# B&R Automation Studio project CombinedLinenSoiledA9KAN (part 6)

```automation-basic
	;bDataValidFlag-> mandatory - TRUE only for last telegram as defined in CAN2 standard..
	bDataValid = FALSE 		; return data's validity status..
	endif
;******CANID421..439******T4******CANID421..439******T4******CANID421..439******T4******CANID421..439******

	;§ ID 421..439 - T4 identified -mandatories..
	if ( BIT_TST(CAN1Data.T_By1,3) AND BIT_TST(CAN1Data.T_By1,4)AND BIT_TST(CAN1Data.T_By1,5)) then

 	; a_usCustomize
		memcpy(adr(a_usOutByteArray[37]) , adr(CAN1Data.T_By0), 1)
			; im By1 liegt das Steuerbyte..
		memcpy(adr(a_usOutByteArray[38]) , adr(CAN1Data.T_By2_By3), 2)
		memcpy(adr(a_usOutByteArray[40]) , adr(CAN1Data.T_By4_By5), 2)
		memcpy(adr(a_usOutByteArray[42]) , adr(CAN1Data.T_By6_By7), 2)

	;bDataValidFlag-> mandatory - TRUE only for last telegram as defined in CAN2 standard..
	bDataValid = TRUE 		; return data's validity status..
	endif
endaction	; 421..439

;******CANID441..459************CANID441..459************CANID441..459************CANID441..459******
action 441..459:

;******CANID441..459******T1******CANID441..459******T1******CANID441..459******T1******CANID441..459******
	;§ CANID441 - T1 identified -mandatories..
; fetch By2 to get controlByte - the LOWERByte..
if(TARGETInfo_0.DataFormat = 2)then ; motorola..
	uiTemp = CAN1Data.T_By2_By3
	usTemp =  USINT(shr(uiTemp,8))
else ; i386
	usTemp = USINT(CAN1Data.T_By2_By3)
endif
	; WETCANII stamp identified.. + TelNo.1
	if ( NOT(BIT_TST(usTemp,6))AND BIT_TST(usTemp,7) ) then
;	bVorsignalFlusen
		if(BIT_TST(usTemp,0) = 1) then
			a_usOutByteArray[7] = 1
		else
			a_usOutByteArray[7] = 0
		endif
;	bSaugbeladungAktiv					1
		if(BIT_TST(usTemp,1) = 1) then
			a_usOutByteArray[8] = 1
		else
			a_usOutByteArray[8] = 0
		endif
;	bAnforderungFlusen					1
		if(BIT_TST(usTemp,2) = 1) then
			a_usOutByteArray[9] = 1
		else
			a_usOutByteArray[9] = 0
		endif
	;	uiTrocknerrestzeit
		if TARGETInfo_0.DataFormat = 2 then ; motorola
			a_usOutByteArray[0] = CAN1Data.T_By0
			a_usOutByteArray[1] = CAN1Data.T_By1
		else if TARGETInfo_0.DataFormat = 1 then ; intel
			a_usOutByteArray[0] = CAN1Data.T_By1
			a_usOutByteArray[1] = CAN1Data.T_By0
		else
		 	uiStatus = TARGETInfo_0.status
		endif
	bDataValid = FALSE ; return data's validity status..
	endif
;******CANID441..459******T2******CANID441..459******T2******CANID441..459******T2******CANID441..459******
	;§ CANID441 - T2 identified -mandatories..

	; WETCANII stamp identified.. + TelNo.2
	if (BIT_TST(usTemp,6)AND BIT_TST(usTemp,7) ) then

		memcpy(adr(a_usOutByteArray[10]), adr(CAN1Data.T_By0),2)
		memcpy(adr(a_usOutByteArray[13]), adr(CAN1Data.T_By4_By5),4)

		usTemp2 =  0
		if TARGETInfo_0.DataFormat = 2 then ; motorola
			usTemp2 = USINT(CAN1Data.T_By2_By3) ; ###HO/UM 130509 V3.3.1
 			memcpy(adr(a_usOutByteArray[12]), adr(usTemp2),1)
		else if TARGETInfo_0.DataFormat = 1 then ; intel
			usTemp2 = USINT(shr(CAN1Data.T_By2_By3,8))
			memcpy(adr(a_usOutByteArray[12]), adr(usTemp2),1)
		else
		 	uiStatus = TARGETInfo_0.status
		endif
	;bDataValidFlag-> mandatory - TRUE only for last telegram as defined in CAN2 standard..
	bDataValid = TRUE 			; return data's validity status..
	endif
endaction ; 441..459

; ###HO-250107 case mittig aufgeteilt -
elseaction:
   	uiStatus = 110
endaction
endcase
RAUS_HIER2:
if uiStatus = 110 then
	; hier weitermachen: zweiten Teil des case durchgehen
else
	; es wurde bereits ein case gefunden - raus hier..
	goto RAUS_HIER3
endif
case udCanID of

action 480:
;******CANID480******T1******CANID480******T1******CANID480******T1******CANID480******T1******CANID480******T1******
; ID 480 - T1 identified -mandatories..
	if (NOT(BIT_TST(CAN1Data.T_By0,5)) AND NOT(BIT_TST(CAN1Data.T_By0,6)) AND BIT_TST(CAN1Data.T_By0,7)) then
;------------------By 0-----------------------------
; 	bBereit
		if(BIT_TST(CAN1Data.T_By0,0) = 1) then
			a_usOutByteArray[0] = 1
		else
			a_usOutByteArray[0] = 0
		endif
; 	bBeladebereit
		if(BIT_TST(CAN1Data.T_By0,1) = 1) then
			a_usOutByteArray[2] = 1
		else
			a_usOutByteArray[2] = 0
		endif
; 	bBeladungAktiv
		if(BIT_TST(CAN1Data.T_By0,2) = 1) then
			a_usOutByteArray[3] = 1
		else
			a_usOutByteArray[3] = 0
		endif
; 	bStoerung
		if(BIT_TST(CAN1Data.T_By0,3) = 1) then
			a_usOutByteArray[4] = 1
		else
			a_usOutByteArray[4] = 0
		endif
; 	bBeladeanfHalbauto
		if(BIT_TST(CAN1Data.T_By0,4) = 1) then
			a_usOutByteArray[5] = 1
		else
			a_usOutByteArray[5] = 0
		endif
;------------------By 1-----------------------------
;	bBeladeabbruch
		if(BIT_TST(CAN1Data.T_By1,0) = 1) then
			a_usOutByteArray[7] = 1
		else
			a_usOutByteArray[7] = 0
		endif
; 	bFreigabeBeladung
		if(BIT_TST(CAN1Data.T_By1,1) = 1) then
			a_usOutByteArray[8] = 1
		else
			a_usOutByteArray[8] = 0
		endif
; 	bDurchschleusenStart
		if(BIT_TST(CAN1Data.T_By1,2) = 1) then
			a_usOutByteArray[9] = 1
		else
			a_usOutByteArray[9] = 0
		endif
;	bNotAusAero
		if(BIT_TST(CAN1Data.T_By1,3) = 1) then
			a_usOutByteArray[1] = 1
		else
			a_usOutByteArray[1] = 0
		endif
;	bBeladepause
		if(BIT_TST(CAN1Data.T_By1,4) = 1) then
			a_usOutByteArray[6] = 1
		else
			a_usOutByteArray[6] = 0
		endif
; Redundanzen b1-4
		if(BIT_TST(CAN1Data.T_By1,5) = 1) then
			a_usOutByteArray[25] = 1
		else
			a_usOutByteArray[25] = 0
		endif
		if(BIT_TST(CAN1Data.T_By1,6) = 1) then
			a_usOutByteArray[26] = 1
		else
			a_usOutByteArray[26] = 0
		endif
		if(BIT_TST(CAN1Data.T_By1,7) = 1) then
			a_usOutByteArray[27] = 1
		else
			a_usOutByteArray[27] = 0
		endif
; udPostennummer
			uiShr8 = shr(CAN1Data.T_By2_By3,8)
		a_usOutByteArray[14] = USINT(uiShr8)
		a_usOutByteArray[15] = USINT(CAN1Data.T_By2_By3)
			uiShr8 = shr(CAN1Data.T_By4_By5,8)
		a_usOutByteArray[16] = USINT(uiShr8)
		a_usOutByteArray[17] = USINT(CAN1Data.T_By4_By5)
; uiGewicht
			uiShr8 = shr(CAN1Data.T_By6_By7,8)
		a_usOutByteArray[22] = USINT(uiShr8)
		a_usOutByteArray[23] = USINT(CAN1Data.T_By6_By7)

	;bDataValidFlag-> mandatory - TRUE only for last telegram as defined in CAN2 standard..
	bDataValid = FALSE 								; return data's validity status..
	endif
;******CANID480******T2******CANID480******T2******CANID480******T2******CANID480******T2******CANID480******

	; CANID480 - T2 identified -mandatories..
	if (BIT_TST(CAN1Data.T_By0,5) AND NOT(BIT_TST(CAN1Data.T_By0,6)) AND BIT_TST(CAN1Data.T_By0,7)) then
; bProgKat
		if(BIT_TST(CAN1Data.T_By0,0) = 1) then
			a_usOutByteArray[10] = 1
		else
			a_usOutByteArray[10] = 0
		endif

; Redundanzen -> T2-By0 - bit1..4
		if(BIT_TST(CAN1Data.T_By0,1) = 1) then
			a_usOutByteArray[28] = 1
		else
			a_usOutByteArray[28] = 0
		endif
		if(BIT_TST(CAN1Data.T_By0,2) = 1) then
			a_usOutByteArray[29] = 1
		else
			a_usOutByteArray[29] = 0
		endif
		if(BIT_TST(CAN1Data.T_By0,3) = 1) then
			a_usOutByteArray[30] = 1
		else
			a_usOutByteArray[30] = 0
		endif
		if(BIT_TST(CAN1Data.T_By0,4) = 1) then
			a_usOutByteArray[31] = 1
		else
			a_usOutByteArray[31] = 0
		endif
; usReserve1
		a_usOutByteArray[24] = CAN1Data.T_By1

; uiProgKat
			uiShr8 = shr(CAN1Data.T_By2_By3,8)
		a_usOutByteArray[12] = USINT(uiShr8)
		a_usOutByteArray[13] = USINT(CAN1Data.T_By2_By3)
; udKundennummer
			uiShr8 = shr(CAN1Data.T_By4_By5,8)
		a_usOutByteArray[18] = USINT(uiShr8)
		a_usOutByteArray[19] = USINT(CAN1Data.T_By4_By5)
			uiShr8 = shr(CAN1Data.T_By6_By7,8)
		a_usOutByteArray[20] = USINT(uiShr8)
		a_usOutByteArray[21] = USINT(CAN1Data.T_By6_By7)

	;bDataValidFlag-> mandatory - TRUE only for last telegram as defined in CAN2 standard..
	bDataValid = FALSE 		; return data's validity status..
	endif
;******CANID480******T3******CANID480******T3******CANID480******T3******CANID480******T3******CANID480******

	; CANID480 - T3 identified -mandatories..
	if (NOT(BIT_TST(CAN1Data.T_By0,5)) AND BIT_TST(CAN1Data.T_By0,6) AND BIT_TST(CAN1Data.T_By0,7)) then

	; Redundanzen -> T3-By0 - bit1..2 - bit3..4 nicht verwendet..
		if(BIT_TST(CAN1Data.T_By0,0) = 1) then
			a_usOutByteArray[32] = 1
		else
			a_usOutByteArray[32] = 0
		endif
		if(BIT_TST(CAN1Data.T_By0,1) = 1) then
			a_usOutByteArray[33] = 1
		else
			a_usOutByteArray[33] = 0
		endif

	; a_usCustomize
		memcpy(adr(a_usOutByteArray[34]) , adr(CAN1Data.T_By1), 1)
		memcpy(adr(a_usOutByteArray[35]) , adr(CAN1Data.T_By2_By3), 2)
		memcpy(adr(a_usOutByteArray[37]) , adr(CAN1Data.T_By4_By5), 2)
		memcpy(adr(a_usOutByteArray[39]) , adr(CAN1Data.T_By6_By7), 2)

	;bDataValidFlag-> mandatory - TRUE only for last telegram as defined in CAN2 standard..
	bDataValid = TRUE 		; return data's validity status..
	endif
endaction ; 480

action 481:
;******CANID481******T1******CANID481******T1******CANID481******T1******CANID481******T1******CANID481******T1******
; ID 481 - T1 identified -mandatories..
	if (NOT(BIT_TST(CAN1Data.T_By0,5)) AND NOT(BIT_TST(CAN1Data.T_By0,6)) AND BIT_TST(CAN1Data.T_By0,7)) then

; bBereit
		if(BIT_TST(CAN1Data.T_By0,0) = 1) then
			a_usOutByteArray[0] = 1
		else
			a_usOutByteArray[0] = 0
		endif
; bBeladeanfAuto
		if(BIT_TST(CAN1Data.T_By0,1) = 1) then
			a_usOutByteArray[2] = 1
		else
			a_usOutByteArray[2] = 0
		endif
; bStoerung
		if(BIT_TST(CAN1Data.T_By0,2) = 1) then
			a_usOutByteArray[3] = 1
		else
			a_usOutByteArray[3] = 0
		endif
; bAnlagenstrgHalbauto
		if(BIT_TST(CAN1Data.T_By0,3) = 1) then
			a_usOutByteArray[4] = 1
		else
			a_usOutByteArray[4] = 0
		endif
; bAnlagenStrgAuto
		if(BIT_TST(CAN1Data.T_By0,4) = 1) then
			a_usOutByteArray[5] = 1
		else
			a_usOutByteArray[5] = 0
		endif
; Redundanzen b1-4
		if(BIT_TST(CAN1Data.T_By1,4) = 1) then
			a_usOutByteArray[23] = 1
		else
			a_usOutByteArray[23] = 0
		endif
		if(BIT_TST(CAN1Data.T_By1,5) = 1) then
			a_usOutByteArray[24] = 1
		else
			a_usOutByteArray[24] = 0
		endif
		if(BIT_TST(CAN1Data.T_By1,6) = 1) then
			a_usOutByteArray[25] = 1
		else
			a_usOutByteArray[25] = 0
		endif
		if(BIT_TST(CAN1Data.T_By1,7) = 1) then
			a_usOutByteArray[26] = 1
		else
			a_usOutByteArray[26] = 0
		endif
; bDurchschleusen
		if(BIT_TST(CAN1Data.T_By1,0) = 1) then
			a_usOutByteArray[7] = 1
		else
			a_usOutByteArray[7] = 0
		endif
; bFreigabeDurchschl
		if(BIT_TST(CAN1Data.T_By1,1) = 1) then
			a_usOutByteArray[8] = 1
		else
			a_usOutByteArray[8] = 0
		endif
; bNotAusAnlagenStrg
		if(BIT_TST(CAN1Data.T_By1,2) = 1) then
			a_usOutByteArray[1] = 1
		else
			a_usOutByteArray[1] = 0
		endif
; bPauseAktiv
		if(BIT_TST(CAN1Data.T_By1,3) = 1) then
			a_usOutByteArray[6] = 1
		else
			a_usOutByteArray[6] = 0
		endif
; udPostennummer
			uiShr8 = shr(CAN1Data.T_By2_By3,8)
		a_usOutByteArray[18] = USINT(uiShr8)
		a_usOutByteArray[19] = USINT(CAN1Data.T_By2_By3)
			uiShr8 = shr(CAN1Data.T_By4_By5,8)
		a_usOutByteArray[20] = USINT(uiShr8)
		a_usOutByteArray[21] = USINT(CAN1Data.T_By4_By5)
; uiGewicht
			uiShr8 = shr(CAN1Data.T_By6_By7,8)
		a_usOutByteArray[12] = USINT(uiShr8)
		a_usOutByteArray[13] = USINT(CAN1Data.T_By6_By7)

	;bDataValidFlag-> mandatory - TRUE only for last telegram as defined in CAN2 standard..
	bDataValid = FALSE 								; return data's validity status..

	endif
;******CANID481******T2******CANID481******T2******CANID481******T2******CANID481******T2******CANID481******

	; CANID481 - T2 identified -mandatories..
	if (BIT_TST(CAN1Data.T_By0,5) AND NOT(BIT_TST(CAN1Data.T_By0,6)) AND BIT_TST(CAN1Data.T_By0,7)) then
; bProgKat
		if(BIT_TST(CAN1Data.T_By0,0) = 1) then
			a_usOutByteArray[9] = 1
		else
			a_usOutByteArray[9] = 0
		endif
; Redundanzen T2By0 /b6-10
		if(BIT_TST(CAN1Data.T_By0,1) = 1) then
			a_usOutByteArray[27] = 1
		else
			a_usOutByteArray[27] = 0
		endif
		if(BIT_TST(CAN1Data.T_By0,2) = 1) then
			a_usOutByteArray[28] = 1
		else
			a_usOutByteArray[28] = 0
		endif
		if(BIT_TST(CAN1Data.T_By0,3) = 1) then
			a_usOutByteArray[29] = 1
		else
			a_usOutByteArray[29] = 0
		endif
		if(BIT_TST(CAN1Data.T_By0,4) = 1) then
			a_usOutByteArray[30] = 1
		else
			a_usOutByteArray[30] = 0
		endif
; usReserve1
		a_usOutByteArray[22] = CAN1Data.T_By1
; uiProgKat
			uiShr8 = shr(CAN1Data.T_By2_By3,8)
		a_usOutByteArray[10] = USINT(uiShr8)
		a_usOutByteArray[11] = USINT(CAN1Data.T_By2_By3)
; udKundennummer
			uiShr8 = shr(CAN1Data.T_By4_By5,8)
		a_usOutByteArray[14] = USINT(uiShr8)
		a_usOutByteArray[15] = USINT(CAN1Data.T_By4_By5)
			uiShr8 = shr(CAN1Data.T_By6_By7,8)
		a_usOutByteArray[16] = USINT(uiShr8)
		a_usOutByteArray[17] = USINT(CAN1Data.T_By6_By7)

	;bDataValidFlag-> mandatory - TRUE only for last telegram as defined in CAN2 standard..
	bDataValid = FALSE 		; return data's validity status..
	endif

;******CANID481******T3******CANID481******T3******CANID481******T3******CANID481******T3******CANID481******

	; CANID481 - T3 identified -mandatories..
	if (NOT(BIT_TST(CAN1Data.T_By0,5)) AND BIT_TST(CAN1Data.T_By0,6) AND BIT_TST(CAN1Data.T_By0,7)) then

	; Redundanzen bR9..10
		if(BIT_TST(CAN1Data.T_By0,1) = 1) then
			a_usOutByteArray[31] = 1
		else
			a_usOutByteArray[31] = 0
		endif
		if(BIT_TST(CAN1Data.T_By0,2) = 1) then
			a_usOutByteArray[32] = 1
		else
			a_usOutByteArray[32] = 0
		endif

	; a_usCustomize
		memcpy(adr(a_usOutByteArray[33]) , adr(CAN1Data.T_By1), 1)
		memcpy(adr(a_usOutByteArray[34]) , adr(CAN1Data.T_By2_By3), 2)
		memcpy(adr(a_usOutByteArray[36]) , adr(CAN1Data.T_By4_By5), 2)
		memcpy(adr(a_usOutByteArray[38]) , adr(CAN1Data.T_By6_By7), 2)

	;bDataValidFlag-> mandatory - TRUE only for last telegram as defined in CAN2 standard..
	bDataValid = TRUE 		; return data's validity status..
	endif
endaction ; 481

;********************************************************************************************************
;********************************************************************************************************
; add new Obj types here..
;********************************************************************************************************
;********************************************************************************************************

elseaction:
	uiStatus = 110
endaction

endcase ; udCanID

RAUS_HIER3:

END_FUNCTION_BLOCK
```

#### _Seti386CAN2TypeToCAN1Type.ab
```automation-basic
FUNCTION_BLOCK _Seti386CAN2TypeToCAN1Type
;********************************************************************************************************
; * Implementation of _Seti386CAN2TypeToCAN1Type
;********************************************************************************************************
; * version 		1.1.0
; * last change		sep, 12th, 2005
; * by				H.O.
;********************************************************************************************************
;********************************************************************************************************
; 	-> 	pCAN2Data			.. pointer to CAN2 structure that contains data to read or write
; 	-> 	iTelegramIndex		.. telegram index exctractet from received / broadcasted telegram
; 		pCAN1Data 		->	.. return the address of CAN1 struct
;********************************************************************************************************
; V1.1.0 ###HO  - 120905
;	* 5th tel added
;********************************************************************************************************

; set local pointer to incoming CAN2 uni structure
pLocalCAN2UniData access (pCAN2Data)
LocalCAN2UniData = pLocalCAN2UniData

; create CAN1 telegram from CAN2 te structure passed in..
case iTelegramIndex of

	action 1:
		LocalCAN1Data.T_By0 	= LocalCAN2UniData.T1_By0
		LocalCAN1Data.T_By1 	= LocalCAN2UniData.T1_By1

		uiShiftUPPERWord 		= shr(LocalCAN2UniData.T1_By2_By3,8) ; move UPPER byte to the right
		uiShiftLOWERWord 		= shl(LocalCAN2UniData.T1_By2_By3,8) ; move LOWER byte to the left
		LocalCAN1Data.T_By2_By3 = uiShiftUPPERWord + uiShiftLOWERWord ; now uiShiftWord contains LocalCAN2UniData.T1_By2_By3 in reverse order

		uiShiftUPPERWord 		= shr(LocalCAN2UniData.T1_By4_By5,8) ; move UPPER byte to the right
		uiShiftLOWERWord 		= shl(LocalCAN2UniData.T1_By4_By5,8) ; move LOWER byte to the left
		LocalCAN1Data.T_By4_By5 = uiShiftUPPERWord + uiShiftLOWERWord ; now uiShiftWord contains LocalCAN2UniData.T1_By2_By3 in reverse order

		uiShiftUPPERWord 		= shr(LocalCAN2UniData.T1_By6_By7,8) ; move UPPER byte to the right
		uiShiftLOWERWord 		= shl(LocalCAN2UniData.T1_By6_By7,8) ; move LOWER byte to the left
		LocalCAN1Data.T_By6_By7 = uiShiftUPPERWord + uiShiftLOWERWord ; now uiShiftWord contains LocalCAN2UniData.T1_By2_By3 in reverse order
	endaction
		action 2:
		LocalCAN1Data.T_By0 	= LocalCAN2UniData.T2_By0
		LocalCAN1Data.T_By1 	= LocalCAN2UniData.T2_By1

		uiShiftUPPERWord 		= shr(LocalCAN2UniData.T2_By2_By3,8) ; move UPPER byte to the right
		uiShiftLOWERWord 		= shl(LocalCAN2UniData.T2_By2_By3,8) ; move LOWER byte to the left
		LocalCAN1Data.T_By2_By3 = uiShiftUPPERWord + uiShiftLOWERWord ; now uiShiftWord contains LocalCAN2UniData.T1_By2_By3 in reverse order

		uiShiftUPPERWord 		= shr(LocalCAN2UniData.T2_By4_By5,8) ; move UPPER byte to the right
		uiShiftLOWERWord 		= shl(LocalCAN2UniData.T2_By4_By5,8) ; move LOWER byte to the left
		LocalCAN1Data.T_By4_By5 = uiShiftUPPERWord + uiShiftLOWERWord ; now uiShiftWord contains LocalCAN2UniData.T1_By2_By3 in reverse order

		uiShiftUPPERWord 		= shr(LocalCAN2UniData.T2_By6_By7,8) ; move UPPER byte to the right
		uiShiftLOWERWord 		= shl(LocalCAN2UniData.T2_By6_By7,8) ; move LOWER byte to the left
		LocalCAN1Data.T_By6_By7 = uiShiftUPPERWord + uiShiftLOWERWord ; now uiShiftWord contains LocalCAN2UniData.T1_By2_By3 in reverse order
	endaction
		action 3:
		LocalCAN1Data.T_By0 	= LocalCAN2UniData.T3_By0
		LocalCAN1Data.T_By1 	= LocalCAN2UniData.T3_By1

		uiShiftUPPERWord 		= shr(LocalCAN2UniData.T3_By2_By3,8) ; move UPPER byte to the right
		uiShiftLOWERWord 		= shl(LocalCAN2UniData.T3_By2_By3,8) ; move LOWER byte to the left
		LocalCAN1Data.T_By2_By3 = uiShiftUPPERWord + uiShiftLOWERWord ; now uiShiftWord contains LocalCAN2UniData.T1_By2_By3 in reverse order

		uiShiftUPPERWord 		= shr(LocalCAN2UniData.T3_By4_By5,8) ; move UPPER byte to the right
		uiShiftLOWERWord 		= shl(LocalCAN2UniData.T3_By4_By5,8) ; move LOWER byte to the left
		LocalCAN1Data.T_By4_By5 = uiShiftUPPERWord + uiShiftLOWERWord ; now uiShiftWord contains LocalCAN2UniData.T1_By2_By3 in reverse order

		uiShiftUPPERWord 		= shr(LocalCAN2UniData.T3_By6_By7,8) ; move UPPER byte to the right
		uiShiftLOWERWord 		= shl(LocalCAN2UniData.T3_By6_By7,8) ; move LOWER byte to the left
		LocalCAN1Data.T_By6_By7 = uiShiftUPPERWord + uiShiftLOWERWord ; now uiShiftWord contains LocalCAN2UniData.T1_By2_By3 in reverse order
	endaction
		action 4:
		LocalCAN1Data.T_By0 	= LocalCAN2UniData.T4_By0
		LocalCAN1Data.T_By1 	= LocalCAN2UniData.T4_By1

		uiShiftUPPERWord 		= shr(LocalCAN2UniData.T4_By2_By3,8) ; move UPPER byte to the right
		uiShiftLOWERWord 		= shl(LocalCAN2UniData.T4_By2_By3,8) ; move LOWER byte to the left
		LocalCAN1Data.T_By2_By3 = uiShiftUPPERWord + uiShiftLOWERWord ; now uiShiftWord contains LocalCAN2UniData.T1_By2_By3 in reverse order

		uiShiftUPPERWord 		= shr(LocalCAN2UniData.T4_By4_By5,8) ; move UPPER byte to the right
		uiShiftLOWERWord 		= shl(LocalCAN2UniData.T4_By4_By5,8) ; move LOWER byte to the left
		LocalCAN1Data.T_By4_By5 = uiShiftUPPERWord + uiShiftLOWERWord ; now uiShiftWord contains LocalCAN2UniData.T1_By2_By3 in reverse order

		uiShiftUPPERWord 		= shr(LocalCAN2UniData.T4_By6_By7,8) ; move UPPER byte to the right
		uiShiftLOWERWord 		= shl(LocalCAN2UniData.T4_By6_By7,8) ; move LOWER byte to the left
		LocalCAN1Data.T_By6_By7 = uiShiftUPPERWord + uiShiftLOWERWord ; now uiShiftWord contains LocalCAN2UniData.T1_By2_By3 in reverse order
	endaction
	action 5:
		LocalCAN1Data.T_By0 	= LocalCAN2UniData.T5_By0
		LocalCAN1Data.T_By1 	= LocalCAN2UniData.T5_By1

		uiShiftUPPERWord 		= shr(LocalCAN2UniData.T5_By2_By3,8) ; move UPPER byte to the right
		uiShiftLOWERWord 		= shl(LocalCAN2UniData.T5_By2_By3,8) ; move LOWER byte to the left
		LocalCAN1Data.T_By2_By3 = uiShiftUPPERWord + uiShiftLOWERWord ; now uiShiftWord contains LocalCAN2UniData.T1_By2_By3 in reverse order

		uiShiftUPPERWord 		= shr(LocalCAN2UniData.T5_By4_By5,8) ; move UPPER byte to the right
		uiShiftLOWERWord 		= shl(LocalCAN2UniData.T5_By4_By5,8) ; move LOWER byte to the left
		LocalCAN1Data.T_By4_By5 = uiShiftUPPERWord + uiShiftLOWERWord ; now uiShiftWord contains LocalCAN2UniData.T1_By2_By3 in reverse order

		uiShiftUPPERWord 		= shr(LocalCAN2UniData.T5_By6_By7,8) ; move UPPER byte to the right
		uiShiftLOWERWord 		= shl(LocalCAN2UniData.T5_By6_By7,8) ; move LOWER byte to the left
		LocalCAN1Data.T_By6_By7 = uiShiftUPPERWord + uiShiftLOWERWord ; now uiShiftWord contains LocalCAN2UniData.T1_By2_By3 in reverse order
	endaction
endcase

; pass pointer to CAN1 telegram to output..
pCAN1Data = ADR(LocalCAN1Data)

;********************************************************************************************************
;********************************************************************************************************
END_FUNCTION_BLOCK
```

#### _swapUINT.ab
```automation-basic
FUNCTION _swapUINT
;*************************************************************************************
(* Implementation of _swapUINT *)
;*************************************************************************************
;  Identisch CONVERT::swapUINT -die macht aber Streit beim Wechsel zw. m68k und i386 !
;*************************************************************************************
usHIGHERBYTE = USINT(shr(uiIn,8))
usLOWERBYTE  = USINT(uiIn)

_swapUINT = usLOWERBYTE*256 + usHIGHERBYTE
;*************************************************************************************
END_FUNCTION
```

#### _version.ab
```automation-basic
FUNCTION_BLOCK _version
;******************************************************************
(* Implementation of _version *)
;******************************************************************
strcpy(adr(szVersion ),"V3.6.2")
uiBuild = 00000 ;  - 170112 - 1230
;******************************************************************
; History
; -------
; V3.6.2 - ###HO - 170112
;	*  Korrektur COB306.uiGew /.bUebergabest /.bNotAusAero
;	*  Korrektur COB316.bBereit
;	*  Korrektur COB371.a_usCustom /.bBereit
; V3.6.1 - ###HO - 160112
;	*  Korrektur: Letztes Einzeltel. 306,316,361..,371.. ohne Inhalt
;		* COB306 Uebergabestörung++ / a_usCustomize++ lt. TIS 2003-07g V1.1.0
;		* COB316 a_usCustomize++ lt. TIS 2003-07g V1.1.0
;		* 361..369 a_uscustomize++ / bBereit ++ lt. TIS 2003-07k V1.1.0
;		* 371..379 a_uscustomize++ / bBereit ++ lt. TIS 2003-07k V1.1.0
; V3.6.0 - ###HO - 120210
;	* COB120 auch für ID 150,160,170,180,190
;	* COB121 auch für ID 151,161,171,181,191
; V3.5.0 - ###HO - 050210
;	* COB301.Entladeueberwachung ++
; V3.4.0 - ###HO - 211209
;	* COB 110 + 111 neu (Test i386 ok, todo: m68k)
; V3.3.2 - ###HO - 130509
;	* WARNUNGEN nicht verw. Var entfernt
; V3.3.1 - ###HO - 130509
;	* SetCAN1TypeToByteArray::Korrektur 4x Compilerwarnung durch BuR UM
; V3.3.0 - ###HO - 140409
;	* COB311.StartPresse
;	* COB211.SicherhTuer
;	* COB211.StartbefAnPT
; V3.2.3 - ###HO - 070308
; 	* COB301.LS_Bandende ++
; 	* COB301.bNotAus --
; 	* COB311.SchutzgitterOffen ++
; 	* COB252.SperreBereich ++
; V3.2.2 - ###HO - 111007
; 	* _SetCAN2COBTypeToCAN2Type::COB211.usFehlerZweiteEW
; 	* _SetCAN1TypeToByteArray:: Korrektur Lesen von 211.bStartDesinfektion, 211.bStartSpuelen, 211.bEndeSpuelen
; V3.2.1 - ###hcs/HO - 101007
; 	COB_ID130und140 und COB_ID131und141 entfernt - stattdessen Neudefinition:
; 		* COB 130 und COB140 wie COB120
;		* COB131 und COB141 wie COB121
; V3.2.0 - ###HO - 040907
;	* COB251.bBeladestart
;		* _SetCAN2COBTypeToCAN2Type
;		* _SetCAN1TypeToByteArray
;		* _ConvertDataToi386
;	* COBs 261,262 hinzugefügt
; 	* neu: COB301bis304, COB311bis314, COB251u253u255, COB252u254u256, COB351bis354
;	* obsolet/umbenannt (s.o.): COB301, COB351, COB251, COB252
; V3.1.2 - ###HO - 250107
;	* _SetCAN2COBTypeToCAN2Type + _SetCAN1TypeToByteArray ::Sprung >32k (MyCheck) beseitigt
; V3.1.1 - ###HO - 110107
;	* _SetCAN2COBTypeToCAN2Type:351 lt. TIS 07j)-V1.4.3
; V3.1.0 - ###HO - 141206
;	* COBs 126,128 (=COB120) und 127,129 (=COB121) hinzugefügt
; V3.0.9 - ###HO - 260106
;	* _SetCAN2COBTypeToCAN2Type + _SetCAN1TypeToByteArray::COB231.Reserve1+2
; V3.0.8 - ###HO - 21.11.2005
;	* _SetCAN2COBTypeToCAN2Type::LocalCOB_Typ_251 -> LocalCOB_Typ_253,LocalCOB_Typ_255,LocalCOB_Typ_257
; V3.0.7 - ###HO - 17.11.2005
;	* Read:COB251=253=255=257
;	* Wrt: COB252=254=256=258
;	* _GetNumberOfCan1Tels::COB254,256,258:: 2->3
;	* _SetCAN2COBTypeToCAN2Type::COB253,255,257::LocalCAN2Data.T2_By0,4
; V3.0.6 - ###HO - 21.10.2005
;	* _SetCAN2COBTypeToCAN2Type::COB_ID421bis439 erweitert für IDs 422..439
; V3.0.5 - ###HO - 14.10.2005
;	* _SetCAN1TypeToByteArray::COB201.uiProgrammKategorie - Alignmentbyte auf xx[5]..
; V3.0.4 - ###HO - 06.10.2005
; 	* a_usCustomize für COBs 301,311,221,231,201,211,209,219
; V3.0.3 - ###HO - 05.10.2005
;	* COB_ID211.bSchiebeimpulsWETShuttle ersetzt durch bSchiebeimpSpbPreXOR_WETShuttle lt. TIS 2003_07c) V1.1.1
; V3.0.2 - ###HO - 19.09.2005
;	* Can2Init().doMemType
; V3.0.0 - ###HO - 12.09.2005
;	* COBxxx.a_usCustomize[0..6] hinzugefügt
;	* COBs 307+317 neu
; V2.1.5 - ###HO - 31.08.2005
;	* Ergänzung Hilfe COB441
;	* Aktualisierung Datentypen ‚COB_ID401bis419’ + ‚COB_ID441bis459’ TIS2003-7h nach V1.2.2b
;V2.1.4 ###HO - 17.02.2005
;·      CAN2Init(): ‚20613’ für ‚usUniqueIDCAN2Init’ > 9
; V2.1.3 ###HO - 110205
; 	* '_SetCAN1TypeToByteArray':: Autoerkennung: Lesen COB120::2oder4Tels
; 	* 'CAN2RW':: Autoerkennung: Schreiben COB120::2oder4Tels
; V2.1.2 ###HO - 070205
;	* V2.1.1 auch für m68k
; V2.1.1 ###HO
; 	* Korrektur Bezeichner szCAN2Write/ReadDO für DatObjCreate() - sonst status '20601'
;	* Speicher für DOs nach Warmstart wurde nicht wieder freigegeben
;		-> Instanzenabhängige Generierung von DOs anhand UniqueCAN2Init-Handle
; V2.1.0 ###HO	150404
;	* Redundancy support done for COBs: 480,481
; 	* COB130.udKundenummer korrigiert
;	* COB201 Desinfektion ergänzt
;		* bFreigabeDesinfektion, bTankIstLeer, bFreigabeSpuelen, EndeDesinfektion
;	* COB211 Desinfektion ergänzt + bSchiebeimpuls in bSchiebeimpulsWETShuttle umbenannt
;		* bSchiebeimpulsZweiteEntwaess korrigiert
;		* bStartDesinfektion,bEndeSpuelen,bStartSpuelen	hinzugefügt
;	* COB401..419
;		* bProgrammabbruch umbenannt in bVorsignal
;		* bKippsperre ergänzt
;	* COB 421..439
;		* 'bEntlaedt' umbenannt in 'bEntlade'
;		* 'bNotAus' umbenannt in 'bNotAusTrockner
; 	* COB231
;		* usEntladungTrockner 	-> By2 + usTransferZBvorHFB			-> By3
;		* usFehlernummer 		-> By4 +  usTransferZBvorTrockner 	-> By5
;	* COB441..459 hinzugefügt
;	* DO "AdrIC2Prot" replaced by pCAN2Init_ident
;	* enable added
;	* Instance individual DOs generated (!)- mandatory for support of same CANIDs on different CANIFs..
; V 2.0.0 ###HO
;		* COBs 123, 251,252,480,481 added
; 		* COB 122 replaced
; 		* COBs 120,121 modified
; 		* COB 122 number of tels changed from two to four
;		* manually passed size of CANQueue removed - Queuesize always is four now..
; 		* DO "AdrIC2Prot" added to replace OutPara 'p_InitCAN2Protocol'
;		* InPara 'p_InitCAN2Protocol' replaced by DO 'AdrIC2Prot'
; 		* Communication-globalPara 'CAN2Init.iMode' replaced by COB-individual-parameter 'InitCAN2PV.iMode'
; 		* mode by that telegrams have been sent within cycletime changed:
;		* 200ms - exclusively between tels with identical CANID
; 		* all tels of WETCAN2Tel are sent immediately
; V1.00 ###HO -	071003
;		* erste Version
;******************************************************************

END_FUNCTION_BLOCK
```

#### CAN2Init.ab
```automation-basic
FUNCTION_BLOCK CAN2Init
;********************************************************************************************************
;* Implementation of CAN2Init
;********************************************************************************************************
; * version 		3.0.2
; * last change		sep, 19th, 2005
; * by				H.O.
;********************************************************************************************************
; * History:
;***********
; * 3.0.2 	###HO - 190905
; 	* IN doMemType anstatt doUSRRAM
; * V2.1.2	###HO - 070205
;	* V2.1.1 auch für m68k
; * V2.1.1
; 	* Korrektur Bezeichner szCAN2Write/ReadDO für DatObjCreate() - sonst status '20601'
;	* Speicher für DOs nach Warmstart wurde nicht wieder freigegeben
;		-> Instanzenabhängige Generierung von DOs anhand UniqueCAN2Init-Handle
; * V2.1.0
;		* DO "AdrIC2Prot" replaced by pCAN2Init_ident
;		* enable added
;		* instance individual DOs generated
; 			-> mandatory for support of same CANIDs on different CANIFs..
; * V 1.0.0		-> 1st version for AS..
; * V 2.0.0
;		* manually passed size of CANQueue removed - Queuesize always is four now..
; 		* DO "AdrIC2Prot" added to replace OutPara 'p_InitCAN2Protocol'
;********************************************************************************************************
;********************************************************************************************************

if (enable = 0) then
	goto ENDE
endif

; initiate return status of CAN2Init()
uiStatus = 0;  105 ;

; generate identifier for InitDO ...
strcpy(ADR(szInitDO),"CAN2Ini") ; ###HO - 170205 - verkürzt - sonst '20613'
usInitDOInstanceNumber = usUniqueIDCAN2Init
itoa(DINT(usInitDOInstanceNumber), adr(szInitDOInstanceNumber))
; ###HO300904 - "CAN2Init1"
strcat(ADR(szInitDO), adr(szInitDOInstanceNumber))

; create DO with R/W info..
DatObjCreate_InitDO.enable	= 1
DatObjCreate_InitDO.grp		= 0
DatObjCreate_InitDO.pName	= ADR(szInitDO) ; "CAN2Init1"
DatObjCreate_InitDO.len		= uiNumberOfCAN2COBs * sizeof(Local_InitCAN2PV) ; size of DO depends on number of COBs..
DatObjCreate_InitDO.MemType	= doMemType ; doUSRRAM 	; = usrram ist warmstartsicher(!)
DatObjCreate_InitDO.Option	= 1 		; 1-> no crc check..
DatObjCreate_InitDO.pCpyData = adr(pStartAdrDO)	; not in use..
DatObjCreate_InitDO FUB DatObjCreate()
if((uiStatus = 0) and (DatObjCreate_InitDO.status <> 20601))  then
	uiStatus = DatObjCreate_InitDO.status
endif

DatObjInfo(1, ADR(szInitDO), DO_StatInfo, DO_ID, DO_StartAdr, DO_Len, DO_Memtype, DO_Option, DO_ChangeDat )
;***************************************************************************************
; generate identifier for InitDO ...
strcpy(ADR(szCAN2WriteDO),"CAN2Wrt") ; ###HO - 170205 - verkürzt - sonst '20613'
itoa(DINT(usInitDOInstanceNumber), adr(szInitDOInstanceNumber))
;###HO 300904 - strcat('szInitDO',,)
strcat(ADR(szCAN2WriteDO), adr(szInitDOInstanceNumber)) ; addInstNumber to szCAN2WriteDO

DatObjCreate_WriteDO.enable		= 1
DatObjCreate_WriteDO.grp		= 0
DatObjCreate_WriteDO.pName		= adr(szCAN2WriteDO) ; "CAN2Write"
DatObjCreate_WriteDO.len		= uiNumberOfCAN2COBs * sizeof(CAN2Write)
DatObjCreate_WriteDO.MemType	= doMemType ; doUSRRAM
DatObjCreate_WriteDO.Option		= 1
DatObjCreate_WriteDO.pCpyData	= adr(pStartAdrDOCAN2Write)
DatObjCreate_WriteDO FUB DatObjCreate()
if((uiStatus = 0) and (DatObjCreate_WriteDO.status <> 20601))  then
	uiStatus = DatObjCreate_WriteDO.status
endif
DatObjInfo(1, ADR(szCAN2WriteDO), DO_StatInfo, DO_IDCAN2Write, DO_StartAdr, DO_Len, DO_Memtype, DO_Option, DO_ChangeDat )
;***************************************************************************************

; generate identifier for InitDO ...
strcpy(ADR(szCAN2ReadDO),"CAN2Rd") ; ###HO - 170205 - verkürzt - sonst '20613'
itoa(DINT(usInitDOInstanceNumber), adr(szInitDOInstanceNumber))
;###HO 300904 - strcat('szInitDO',,)
strcat(ADR(szCAN2ReadDO), adr(szInitDOInstanceNumber)) ; addInstNumber to szCAN2ReadDO

DatObjCreate_ReadDO.enable		= 1
DatObjCreate_ReadDO.grp			= 0
DatObjCreate_ReadDO.pName		= ADR(szCAN2ReadDO)
DatObjCreate_ReadDO.len			= uiNumberOfCAN2COBs * sizeof(CAN2Read)
DatObjCreate_ReadDO.MemType		= doMemType ; doUSRRAM
DatObjCreate_ReadDO.Option		= 1
DatObjCreate_ReadDO.pCpyData	= adr(pStartAdrDOCAN2Read)
DatObjCreate_ReadDO FUB DatObjCreate()
if((uiStatus = 0) and (DatObjCreate_ReadDO.status <> 20601))  then
	uiStatus = DatObjCreate_ReadDO.status
endif
DatObjInfo(1, adr(szCAN2ReadDO), DO_StatInfo, DO_IDCAN2Read, DO_StartAdr, DO_Len, DO_Memtype, DO_Option, DO_ChangeDat )

;********************************************
; prepare writing to DO
DatObjWrite_InitDO.enable	= 1							; wanna write to DO..
DatObjWrite_InitDO.ident	= DO_ID						; from DOInfo..
DatObjWrite_InitDO.len		= sizeof(Local_InitCAN2PV) 	; size of single DO - former LocalCAN2InitData
;********************************************
DatObjWrite_WriteDO.enable	= 1
DatObjWrite_WriteDO.ident	= DO_IDCAN2Write
DatObjWrite_WriteDO.len		= sizeof(CAN2Write)
;********************************************
DatObjWrite_ReadDO.enable	= 1
DatObjWrite_ReadDO.ident	= DO_IDCAN2Read
DatObjWrite_ReadDO.len		= sizeof(CAN2Read)
;********************************************

; CANOpen() sufficent for CANrd() + CANqwrite()
CANopen_0.enable	= 1
CANopen_0.baud_rate	= 25
CANopen_0.cob_anz	= uiNumberOfCAN2COBs *2
CANopen_0.error_adr	= ADR(ErrAdrNotInUse)
CANopen_0.device	= ADR(szCANInterface)
CANopen_0.info		= 0 ; don't use extd mode of CANCtrl ..
CANopen_0 FUB CANopen()
if(uiStatus = 0) then
	uiStatus = CANopen_0.status
endif
;********************************************

; now -fill DOs with necessarily data
loop iLoopIdx = 0 to (uiNumberOfCAN2COBs -1) do
	memcpy(adr(LocalInitCAN2PV), (pInitCAN2PV + sizeof(LocalInitCAN2PV)*iLoopIdx), sizeof(LocalInitCAN2PV))

	; pass 'InitData' -> '_InitData' ..
	Local_InitCAN2PV.pPVData			= LocalInitCAN2PV.pPVData
	Local_InitCAN2PV.uiObjNr			= LocalInitCAN2PV.uiCANID
	Local_InitCAN2PV.usCommDirection	= LocalInitCAN2PV.usCommDirection
	Local_InitCAN2PV.pEvVar				= LocalInitCAN2PV.pEvVar
	Local_InitCAN2PV.uiCOB_ident		= UINT(iLoopIdx + 900) 	; internal identifier - not in use
	Local_InitCAN2PV.bRunning			= FALSE 				; not in use
	; from V1.1.0 -> COB-individual selection of mode..
	Local_InitCAN2PV.iMode				= LocalInitCAN2PV.iMode

	; check CommDirection to decide whether to initiate a CANqueue() ..
	; initiate for all read operations single CANqueue  - establishing CANQueue only in read direction necessary..
	if (LocalInitCAN2PV.usCommDirection = 0) then		; read to COB..

		; initiate CANqueue for read operation..
		CANqueue_0.enable	= 1
		CANqueue_0.us_ident	= CANopen_0.us_ident
		CANqueue_0.can_id	= LocalInitCAN2PV.uiCANID
		; uiCANqueueSize from V1.0.0 removed -> set to max count of single tels..
		CANqueue_0.size		= 5 ; telegram capacity of queue..
		CANqueue_0 FUB CANqueue()
		if(uiStatus = 0) then
			uiStatus = CANqueue_0.status
			exitif (CANqueue_0.status <> 0)
		endif

		_GetNumberOfCan1Tels_0.pPV		= Local_InitCAN2PV.pPVData
		_GetNumberOfCan1Tels_0.uiObjNr	= Local_InitCAN2PV.uiObjNr
		_GetNumberOfCan1Tels_0 FUB _GetNumberOfCan1Tels()

		; uiCAN_q_ident isn't passed in by user -> created by CANqueue ..
		Local_InitCAN2PV.udCAN_q_ident	= CANqueue_0.q_ident ;

		; write uiObjNr to DO..
		CAN2Read.uiObjNr				= Local_InitCAN2PV.uiObjNr
		CAN2Read.iNumberOfTels			= _GetNumberOfCan1Tels_0.iNumberOfCan1Tels
		CAN2Read.iNumberReceivedTels	= 0

		; reset data of WriteDO
		CAN2Write.bBusy 			= FALSE
		CAN2Write.iNumberOfTels 	= 0
		CAN2Write.iTelsSent			= 0
		CAN2Write.tTimeLastTelSent 	= TIME(0)
		CAN2Write.uiCOB_ident		= iLoopIdx + 900

	else if (LocalInitCAN2PV.usCommDirection = 1) then	; COB is defined as to 'write'
		Local_InitCAN2PV.udCAN_q_ident	= 0	; object to write - no queue established

		; establish DO with CAN2Data of COBs to write..
		_GetNumberOfCan1Tels_0.pPV		= Local_InitCAN2PV.pPVData
		_GetNumberOfCan1Tels_0.uiObjNr	= Local_InitCAN2PV.uiObjNr
		_GetNumberOfCan1Tels_0 FUB _GetNumberOfCan1Tels()

		_SetCAN2COBTypeToCAN2Type_0.p_InitCAN2PV = adr(Local_InitCAN2PV)
		_SetCAN2COBTypeToCAN2Type_0 FUB _SetCAN2COBTypeToCAN2Type()
		; don't read PVs now- actualize process images at runtime..
		; memcpy(adr(CAN2Write.CAN2), _SetCAN2COBTypeToCAN2Type_0.pCAN2DtaUni, sizeof(CAN2Write.CAN2))

		CAN2Write.bBusy 			= FALSE
		CAN2Write.iNumberOfTels 	= _GetNumberOfCan1Tels_0.iNumberOfCan1Tels
		CAN2Write.iTelsSent			= 0
		CAN2Write.tTimeLastTelSent 	= TIME(0)
		CAN2Write.uiCOB_ident		= iLoopIdx + 900

			; reset content of DORead
			CAN2Read.uiObjNr = 0
			loop iLoopIdxTemp = 0 to 49 do  ; ###HO -020905
				CAN2Read.ab_ByteArray[iLoopIdxTemp] = 0
			endloop
	else ; neither read nor write..
		uiStatus = 520
		memcpy(Local_InitCAN2PV.pEvVar,adr(uiStatus),sizeof(uiStatus))
	endif

	DatObjWrite_ReadDO.Offset	= sizeof(CAN2Read) * iLoopIdx
	DatObjWrite_ReadDO.pSource	= adr(CAN2Read)
	DatObjWrite_ReadDO FUB DatObjWrite()
	if(uiStatus = 0) then
		uiStatus = DatObjWrite_ReadDO.status
		exitif (DatObjWrite_ReadDO.status <> 0)
	endif

	; write data to DO..
	DatObjWrite_WriteDO.Offset	= sizeof(CAN2Write) * iLoopIdx
	DatObjWrite_WriteDO.pSource	= adr(CAN2Write)
	DatObjWrite_WriteDO FUB DatObjWrite()
	if(uiStatus = 0) then
		uiStatus = DatObjWrite_WriteDO.status
		exitif (DatObjWrite_WriteDO.status <> 0)
	endif

	; .. and write to InitDO..
	DatObjWrite_InitDO.pSource	= ADR(Local_InitCAN2PV)
	DatObjWrite_InitDO.Offset 	= sizeof(Local_InitCAN2PV) * iLoopIdx
	DatObjWrite_InitDO FUB DatObjWrite()
	if(uiStatus = 0) then
		uiStatus = DatObjWrite_InitDO.status
		exitif (DatObjWrite_InitDO.status <> 0)
	endif
endloop

; now verify protocol data..
if( (uiNumberOfCAN2COBs < 0) or (uiNumberOfCAN2COBs = 0) ) then
	uiStatus = 530
endif

; pass access data to output..
Local_InitCAN2Protocol.AccessInitDO.DO_us_ident  		= DO_ID
Local_InitCAN2Protocol.DoAccessCAN2Write.DO_us_ident 	= DO_IDCAN2Write
Local_InitCAN2Protocol.DOAccessCAN2Read.DO_us_ident 	= DO_IDCAN2Read
Local_InitCAN2Protocol.CAN2DObCount						= uiNumberOfCAN2COBs
Local_InitCAN2Protocol.CANAccess.CANopen_us_ident		= CANopen_0.us_ident
; from V1.1.0 -> param iMode not in use any longer..
Local_InitCAN2Protocol.iMode 							= 111

; assign local data to pointer passed to output.. -> removed from > V1.1.0
; reactivated in V2.1.0
p_InitCAN2Protocol = ADR(Local_InitCAN2Protocol)

; assign handle for CAN2RW()..
pCAN2Init_ident = p_InitCAN2Protocol

;********************************************************************************************************

ENDE:
END_FUNCTION_BLOCK
```

### Data object Logical/ioimgcfg (Simple)

#### ioimgcfg.dat
```
; Automation Studio generated file.
; Each change of the file content causes the deactivation
; of the further automatic actualization of this file by the Automation Studio!
```

### Package Logical/Timestamp - Keeps current timestamp

### Program Logical/Timestamp/zzGetTime (IEC)

#### zzGetTimeCyclic.ab - Cyclic code
```automation-basic
(********************************************************************
 * COPYRIGHT -- HP
 ********************************************************************
 * Program: zzGetTime
 * File: zzGetTimeCyclic.ab
 * Author: treamsbottom
 * Created: June 04, 2014
 ********************************************************************
 * Implementation of program zzGetTime
 ********************************************************************)

PROGRAM _CYCLIC

	GetTimeStamp.enable = TRUE
	GetTimeStamp FUB DTGetTime()
	IF GetTimeStamp.status = ERR_OK THEN
		CurrentTimestamp = GetTimeStamp.DT1
	ENDIF
	D32[78] = UDINT(CurrentTimestamp);

	//Set the current time.
	//DTSetTime(enable, DT1, status)
	setTimeStamp.enable := (D32[79] > 0)
	setTimeStamp.DT1 := DT(D32[79]); 	CAST D32 TO DT
	setTimeStamp FUB DTSetTime()
	IF (setTimeStamp.status =  ERR_OK) THEN
		D32[79] = 0
	ENDIF

END_PROGRAM
```

### Package Logical/Data_BackUp - *Handles all data back up

### Data_BackUp.typ - Global data types
```iecst
(********************************************************************
 * COPYRIGHT -- HP
 ********************************************************************
 * Package: Data_BackUp
 * File: Data_BackUp.typ
 * Author: treamsbottom
 * Created: March 20, 2014
 ********************************************************************
 * Data types of package Data_BackUp
 ********************************************************************)

TYPE
	enum_BackUpAreas :
		(
		eBag,
		eC,
		eD,
		eD32,
		eReportBuffer,
		eRB_Posn,
		eRB_Perm,
		eSQL,
		eRFIDCodes
		);
	Debug_typ : 	STRUCT
		WriteCount_MEM : UDINT;
		ReadCount_MEM : UDINT;
		WriteCount_USB : UDINT;
		ReadCount_USB : UDINT;
		WriteFail_MEM : UDINT;
		ReadFail_MEM : UDINT;
		WriteFail_USB : UDINT;
		ReadFail_USB : UDINT;
	END_STRUCT;
END_TYPE
```

### Data_BackUp.var - Global variables
```iecst
(********************************************************************
 * COPYRIGHT -- HP
 ********************************************************************
 * Package: Data_BackUp
 * File: Data_BackUp.var
 * Author: treamsbottom
 * Created: March 20, 2014
 ********************************************************************
 * Variables of package Data_BackUp
 ********************************************************************)
VAR CONSTANT
	cBackUp_FromSYSROM : USINT := 1;
	cBackUp_FromUSB : USINT := 2;
	cBackUp_StartWithoutRestore : USINT := 10;
END_VAR
```

### Program Logical/Data_BackUp/zzDataStore (IEC) - *Store all data

#### zzDataStore.ab - Implementation code
```automation-basic
(********************************************************************
 * COPYRIGHT -- HP
 ********************************************************************
 * Program: zzDataStore
 * File: zzDataStore.ab
 * Author: treamsbottom
 * Created: March 20, 2014
 ********************************************************************
 * Implementation of program zzDataStore
 ********************************************************************)
;-- V1.01 21-03-2014 First Version-- TR.

PROGRAM _INIT
;Set Global Memtype
MemType = doSYSROM
pUSBDevice = ADR("USBStick")

;Set the Data to be backed up
;Name must be 10 chars max
Backup[0].MemTyp = MemType
Backup[0].DataLength = SIZEOF(Bag)
Backup[0].pData 	= ADR(Bag)
Backup[0].pFileName	= ADR("Bak_Bag")

Backup[1].MemTyp = MemType
Backup[1].DataLength = SIZEOF(C)
Backup[1].pData 	= ADR(C)
Backup[1].pFileName	= ADR("Bak_C")

Backup[2].MemTyp = MemType
Backup[2].DataLength = SIZEOF(D)
Backup[2].pData 	= ADR(D)
Backup[2].pFileName	= ADR("Bak_D")

Backup[3].MemTyp = MemType
Backup[3].DataLength = SIZEOF(D32)
Backup[3].pData 	= ADR(D32)
Backup[3].pFileName	= ADR("Bak_D32")

Backup[4].MemTyp = MemType
Backup[4].DataLength = SIZEOF(ReportBuffer)
Backup[4].pData 	= ADR(ReportBuffer)
Backup[4].pFileName	= ADR("Bak_Report")

Backup[5].MemTyp = MemType
Backup[5].DataLength = SIZEOF(RB_Posn)
Backup[5].pData 	= ADR(RB_Posn)
Backup[5].pFileName	= ADR("Bak_RBPosn")

Backup[6].MemTyp = MemType
Backup[6].DataLength = SIZEOF(RB_Perm)
Backup[6].pData 	= ADR(RB_Perm)
Backup[6].pFileName	= ADR("Bak_RBPerm")

Backup[7].MemTyp = MemType
Backup[7].DataLength = SIZEOF(SQL)
Backup[7].pData 	= ADR(SQL)
Backup[7].pFileName	= ADR("Bak_SQL")

;Backup[8].MemTyp = MemType
;Backup[8].DataLength = SIZEOF(RFIDCode)
;Backup[8].pData 	= ADR(RFIDCode)
;Backup[8].pFileName	= ADR("Bak_RFID")

MaxBackUpAreas = 7

END_PROGRAM

PROGRAM _CYCLIC
IF TestTIM THEN
	memcpy(ADR(D),1,100000)
	TestTIM = FALSE
ENDIF
myMonitorReg = 291 ; D reg to monitor if 0 then stop back up
myUpdateReg	= 292 ; Reply reg from Trackview used to restore data.
myAlarm = 215

Alarm[myAlarm].On	= FALSE
Alarm[myAlarm].Bag 	= 0
Alarm[myAlarm].Name	= 0

CASE eBackup OF
	ACTION eNull:
		IF (D[myUpdateReg] = cBackUp_FromSYSROM) THEN
			;Registers are updated when Read completes
			eBackup = eRead
		ELSE IF (D[myUpdateReg] = cBackUp_FromUSB) THEN
			D[myUpdateReg] = 0
			eBackup = eReadFromUSB
		ELSE IF (D[myUpdateReg] = cBackUp_StartWithoutRestore) THEN
			D[myMonitorReg] = 1
			D[myUpdateReg] = 0
		ELSE
			D[myUpdateReg] = 0
			 IF (D[myMonitorReg] > 0) THEN
				eBackup = eWrite
			ENDIF
		ENDIF
		n = 0
	ENDACTION

	ACTION eWrite: ; Back up perm memory
		BackUp.Enable = TRUE
		BackUp.DataAction = eWrite
		BackUp.DataLength = Backup[n].DataLength
		BackUp.MemType = Backup[n].MemTyp
		BackUp.pData = Backup[n].pData
		BackUp.pFileName = Backup[n].pFileName
		BackUp FUB DataBackUp()
		IF ((BackUp.Status = ERR_OK) OR (BackUp.Status <> ERR_FUB_BUSY)) THEN
			Backup[n].ident = BackUp.CurrentDatFile.ident
			IF (D[myMonitorReg] > 0) THEN
				INC n
				IF (n > MaxBackUpAreas)THEN
					n = 0
					eBackup = eCopyToUSB
				ENDIF
				IF (BackUp.Status = ERR_OK) THEN
					INC Debug.WriteCount_MEM
				ELSE IF (BackUp.Status <> ERR_FUB_BUSY) THEN
					INC Debug.WriteFail_MEM
				ENDIF
			ELSE
				eBackup = eNull
			ENDIF
		ENDIF
	ENDACTION

	ACTION eRead: ; Restore perm memory

		BackUp.Enable = TRUE
		BackUp.DataAction = eRead
		BackUp.DataLength = Backup[n].DataLength
		BackUp.pData = Backup[n].pData
		BackUp.pFileName = Backup[n].pFileName
		BackUp FUB DataBackUp()
		IF ((BackUp.Status = ERR_OK) OR (BackUp.Status <> ERR_FUB_BUSY)) THEN
			Backup[n].ident = BackUp.CurrentDatFile.ident
			INC n
			IF (BackUp.Status = ERR_OK) THEN
				INC Debug.ReadCount_MEM
			ELSE IF (BackUp.Status <> ERR_FUB_BUSY) THEN
				INC Debug.ReadFail_MEM
			ENDIF
			IF (n > MaxBackUpAreas)THEN
				D[myUpdateReg] = 0
				eBackup = eNull
			ENDIF
		ENDIF
	ENDACTION

	ACTION eCopyToUSB: ; Copy all data files to USBStick
		CopytoUSB.Enable = TRUE
		CopytoUSB.pDevice = pUSBDevice
		CopytoUSB.pData = Backup[n].pData
		CopytoUSB.fiLen = Backup[n].DataLength
		CopytoUSB.pFile = Backup[n].pFileName
		CopytoUSB FUB CopyToFileDevice()
		IF CopytoUSB.Status = ERR_OK THEN
			IF (D[myMonitorReg] > 0) THEN
				INC n
				INC Debug.WriteCount_USB
				IF (n > MaxBackUpAreas)THEN
					eBackup = eNull
				ENDIF
			ELSE
				eBackup = eNull
			ENDIF
		ELSE IF CopytoUSB.Status = fiERR_FILE_DEVICE THEN ; File Device doesn't exist go back to writing to SYSROM
			eBackup = eNull
		ELSE IF CopytoUSB.Status <> ERR_FUB_BUSY THEN
			IF (D[myMonitorReg] > 0) THEN
				INC n
				INC Debug.WriteFail_USB
				IF (n > MaxBackUpAreas)THEN
					eBackup = eNull
				ENDIF
			ELSE
				eBackup = eNull
			ENDIF
		ENDIF
	ENDACTION

	ACTION eReadFromUSB:
		ReadFromUSB.Enable = TRUE
		ReadFromUSB.pDevice = pUSBDevice
		ReadFromUSB.pFile = Backup[n].pFileName
		ReadFromUSB.fiLen = Backup[n].DataLength
		ReadFromUSB.pDest = Backup[n].pData
		ReadFromUSB FUB	ReadFromFileDevice()
		IF ReadFromUSB.Status = ERR_OK THEN
			INC n
			INC Debug.ReadCount_USB
			IF (n > MaxBackUpAreas)THEN
				eBackup = eNull
			ENDIF
		ELSE IF ReadFromUSB.Status = fiERR_FILE_DEVICE THEN ; File Device doesn't exist go back to writing to SYSROM
			eBackup = eNull
		ELSE IF  ReadFromUSB.Status <> ERR_FUB_BUSY THEN
			INC n
			INC Debug.ReadFail_USB
			IF (n > MaxBackUpAreas)THEN
				eBackup = eNull
			ENDIF
		ENDIF
	ENDACTION
ENDCASE

IF D[myMonitorReg] = 0 THEN
	Alarm[myAlarm].Name = almBackUpNotRunning
	Alarm[myAlarm].On = TRUE
ENDIF

END_PROGRAM

PROGRAM _EXIT
;Copy all back up files to MemCard

END_PROGRAM
```

#### zzDataStore.var - Local variables
```iecst
(********************************************************************
 * COPYRIGHT -- HP
 ********************************************************************
 * Program: zzDataStore
 * File: zzDataStore.var
 * Author: treamsbottom
 * Created: March 20, 2014
 ********************************************************************
 * Local variables of program zzDataStore
 ********************************************************************)
VAR
	eDataBackup : enum_DataBackup;
	CreateDataFile : DatObjCreate;
	GetFileInfo : DatObjInfo;
	pFile_D : UDINT;
	CurrentDatFile : DatFile_typ;
	WriteData : DatObjWrite;
	ReadData : DatObjRead;
	BackUp : DataBackUp;
	eBackupArea : enum_BackUpAreas;
	Backup : ARRAY[0..9] OF Backup_typ;
	MemType : USINT;
	MaxBackUpAreas : UINT;
	n : UINT;
	eBackup : enum_BackUpState;
	TestTIM : BOOL;
	DataMove : DatObjMove;
	myMonitorReg : UINT;
	myUpdateReg : UINT;
	myAlarm : UINT;
	pUSBDevice : UDINT;
	CopytoUSB : CopyToFileDevice;
	ReadFromUSB : ReadFromFileDevice;
END_VAR
VAR RETAIN
	Debug : Debug_typ;
END_VAR
```

### Library Logical/Data_BackUp/DataBackUp (IEC) - *BackUp and Restore Function
Depends on: DataObj

#### DataSave.ab - *Save Memory to Dat file
```automation-basic
(********************************************************************
 * COPYRIGHT -- HP
 ********************************************************************
 * Library: DataBackUp
 * File: DataSave.ab
 * Author: treamsbottom
 * Created: March 20, 2014
 ********************************************************************
 * Implementation of library DataBackUp
 ********************************************************************)

(* *Save Memory to Dat file *)
FUNCTION_BLOCK DataBackUp
	IF Enable THEN
		IF (Status <> ERR_FUB_BUSY) THEN
		   IF DataAction = eRead THEN
				CurrentDatFile.State = eRead
				eDataBackup = eData_Info
			ELSE IF DataAction = eWrite THEN
				eDataBackup = eData_Create
				CurrentDatFile.State = eWrite
			ENDIF
		ENDIF
		Status = ERR_FUB_BUSY
	ENDIF

	CASE eDataBackup OF
		ACTION eData_DoNothing:
;			CurrentDatFile.ident = 0
;			CurrentDatFile.pDatObjMem = 0
;			CurrentDatFile.len = 0
;			CurrentDatFile.MemType = 0
;			CurrentDatFile.Option = 0
;			CurrentDatFile.ChangeDate = 0
			Status = ERR_OK
		ENDACTION

		ACTION eData_Create:
			CreateDataFile.enable = TRUE
			CreateDataFile.grp = 0
			CreateDataFile.pName = pFileName
			CreateDataFile.len = DataLength
			CreateDataFile.MemType = MemType;doSYSROM
			CreateDataFile.Option = 0; Use CheckSum
			CreateDataFile.pCpyData	= pData
			CreateDataFile	FUB DatObjCreate()
			IF CreateDataFile.status = ERR_OK THEN
				eDataBackup = eData_DoNothing
			ELSE IF CreateDataFile.status = doERR_DUPOBJECT THEN
				eDataBackup = eData_Info
			ELSE IF CreateDataFile.status <> ERR_FUB_BUSY THEN
				Status = CreateDataFile.status
			ENDIF
		ENDACTION

		ACTION eData_Info:
			GetFileInfo.enable = TRUE
			GetFileInfo.pName = pFileName
			GetFileInfo FUB DatObjInfo()
			IF GetFileInfo.status = ERR_OK THEN
				CurrentDatFile.ident = GetFileInfo.ident
				CurrentDatFile.pDatObjMem = GetFileInfo.pDatObjMem
				CurrentDatFile.len = GetFileInfo.len
				CurrentDatFile.MemType = GetFileInfo.MemType
				CurrentDatFile.Option = GetFileInfo.Option
				CurrentDatFile.ChangeDate = GetFileInfo.ChangeDate
				IF CurrentDatFile.State = eRead THEN
					eDataBackup = eData_Read
				ELSE IF	CurrentDatFile.State = eWrite THEN
					eDataBackup = eData_Write
				ENDIF
			ELSE IF GetFileInfo.status <> ERR_FUB_BUSY THEN
				Status = GetFileInfo.status
			ENDIF
		ENDACTION

		ACTION eData_Write:
			WriteData.enable = TRUE
			WriteData.ident = CurrentDatFile.ident
			WriteData.len = DataLength
			WriteData.Offset = 0
			WriteData.pSource = pData
			WriteData FUB DatObjWrite()
			IF WriteData.status = ERR_OK THEN
				Status = ERR_OK
			ELSE IF WriteData.status <> ERR_FUB_BUSY THEN
				Status = WriteData.status
			ENDIF
		ENDACTION

		ACTION eData_Delete:

		ENDACTION

		ACTION eData_Read:
			ReadData.enable = TRUE
			ReadData.ident = CurrentDatFile.ident
			ReadData.len = DataLength
			ReadData.Offset = 0
			ReadData.pDestination = pData
			ReadData FUB DatObjRead()
			IF ReadData.status = ERR_OK THEN
				Status = ERR_OK
			ELSE IF ReadData.status <> ERR_FUB_BUSY THEN
				Status = ReadData.status
			ENDIF
		ENDACTION
	ENDCASE

END_FUNCTION_BLOCK
```

#### CopyToFileDevice.ab - *Write to File. Create if it doesn;t exist
```automation-basic
(********************************************************************
 * COPYRIGHT -- HP
 ********************************************************************
 * Library: DataBackUp
 * File: FileWrite.ab
 * Author: treamsbottom
 * Created: March 24, 2014
 ********************************************************************
 * Implementation of library DataBackUp
 ********************************************************************)

(* *Write to File. Create if it doesn;t exist *)
FUNCTION_BLOCK CopyToFileDevice

IF Enable  THEN
	IF Status <> ERR_FUB_BUSY THEN
		WriteAction = eOpenFile
		Status = ERR_FUB_BUSY
	ENDIF
ENDIF

CASE WriteAction OF
	ACTION eOpenFile:
		OpenFile.enable = TRUE
		OpenFile.mode = fiWRITE_ONLY
		OpenFile.pDevice = pDevice
		OpenFile.pFile = pFile
		OpenFile FUB FileOpen()
		IF OpenFile.status = ERR_OK THEN
			WriteAction = eWriteToFile
			fiIdent = OpenFile.ident
		ELSE IF OpenFile.status = fiERR_FILE_NOT_FOUND THEN
			WriteAction = eCreateFile
		ELSE IF OpenFile.status <> ERR_FUB_BUSY THEN
			Status = OpenFile.status
		ENDIF
	ENDACTION

	ACTION eCreateFile:
		CreateFile.enable = TRUE
		CreateFile.pDevice = pDevice
		CreateFile.pFile = pFile
		CreateFile FUB FileCreate()
		IF CreateFile.status = ERR_OK THEN
			WriteAction = eWriteToFile
			fiIdent = CreateFile.ident
		ELSE IF CreateFile.status <> ERR_FUB_BUSY THEN
			Status = CreateFile.status
		ENDIF
	ENDACTION

	ACTION eWriteToFile:
		WriteFile.enable = TRUE
		WriteFile.ident = fiIdent
		WriteFile.len = fiLen
		WriteFile.offset = 0
		WriteFile.pSrc = pData
		WriteFile FUB FileWrite()
		IF ((WriteFile.status = ERR_OK) OR (WriteFile.status <> ERR_FUB_BUSY)) THEN
			WriteAction = eCloseFile
		ENDIF
	ENDACTION

	ACTION eCloseFile:
		CloseFile.enable = TRUE
		CloseFile.ident = fiIdent
		CloseFile FUB FileClose()
		IF ((CloseFile.status = ERR_OK) OR (CloseFile.status <> ERR_FUB_BUSY)) THEN
			Status = CloseFile.status
		ENDIF
	ENDACTION
ENDCASE

END_FUNCTION_BLOCK
```

#### ReadFromFileDevice.ab - *Open & Read file from File device
```automation-basic
(********************************************************************
 * COPYRIGHT -- HP
 ********************************************************************
 * Library: DataBackUp
 * File: ReadFromFileDevice.ab
 * Author: treamsbottom
 * Created: March 24, 2014
 ********************************************************************
 * Implementation of library DataBackUp
 ********************************************************************)

(* *Open & Read file from File device *)
FUNCTION_BLOCK ReadFromFileDevice
IF Enable  THEN
	IF Status <> ERR_FUB_BUSY THEN
		WriteAction = eOpenFile
		Status = ERR_FUB_BUSY
	ENDIF
ENDIF

CASE WriteAction OF
	ACTION eOpenFile:
		OpenFile.enable = TRUE
		OpenFile.mode = fiREAD_ONLY
		OpenFile.pDevice = pDevice
		OpenFile.pFile = pFile
		OpenFile FUB FileOpen()
		IF OpenFile.status = ERR_OK THEN
			WriteAction = eReadFromFile
			fiIdent = OpenFile.ident
		ELSE IF OpenFile.status <> ERR_FUB_BUSY THEN
			Status = OpenFile.status
		ENDIF
	ENDACTION

	ACTION eReadFromFile:
		ReadFile.enable = TRUE
		ReadFile.ident = fiIdent
		ReadFile.offset = 0
		ReadFile.len = fiLen
		ReadFile.pDest = pDest
		ReadFile FUB FileRead()
		IF ((ReadFile.status = ERR_OK) OR (ReadFile.status <> ERR_FUB_BUSY)) THEN
			WriteAction = eCloseFile
		ENDIF
	ENDACTION

	ACTION eCloseFile:
		CloseFile.enable = TRUE
		CloseFile.ident = fiIdent
		CloseFile FUB FileClose()
		IF ((CloseFile.status = ERR_OK) OR (CloseFile.status <> ERR_FUB_BUSY)) THEN
			Status = CloseFile.status
		ENDIF
	ENDACTION
ENDCASE

END_FUNCTION_BLOCK
```

### Program Logical/SQL/SQLSpeedTest

#### SQLSpeedTestCyclic.ab
```automation-basic
(********************************************************************
 * COPYRIGHT -- HP
 ********************************************************************
 * Program: SQLSpeedTest
 * File: SQLSpeedTestCyclic.ab
 * Author: treamsbottom
 * Created: October 03, 2013
 ********************************************************************
 * Implementation of program SQLSpeedTest
 ********************************************************************)
PROGRAM _INIT
Sql = 0

END_PROGRAM
PROGRAM _CYCLIC

pServer = ADR("10.8.4.200:1433")
pDatabaseName = ADR("SUPDB1")
pUserName = ADR("SUP")
pPassword = ADR("1234")
;	IF pServer <> TestVar THEN
;		INC Break
;		strcpy(ADR(ErrorString),pServer)
;	ENDIF

CASE Sql OF

	ACTION 0:
		SqlConnect.enable = TRUE
		SqlConnect.pServerName = ADR("10.8.4.200:1433")
		SqlConnect.pDatabaseName = ADR("SUPDB1")
		SqlConnect.pUserName = ADR("SUP")
		SqlConnect.pPassword = ADR("1234")
		SqlConnect.databaseSystem = DB_SYSTEM_MS_SQL
		SqlConnect FUB dbConnect()

		IF SqlConnect.status = ERR_OK THEN

			Ident = SqlConnect.connectionIdent
			IF Ident > 0 THEN
				Sql = 1
				INC ConnectionCount
			ENDIF
		ELSE IF SqlConnect.status <> ERR_FUB_BUSY THEN
			IF SqlConnect.connectionIdent <> 0 THEN
				Ident = SqlConnect.connectionIdent
				Sql = 3
			ENDIF
		ELSE IF Ident <> 0 THEN; Connection already made disconnect
			Sql = 2
		ENDIF
	ENDACTION

	ACTION 1:
		SqlExecute.enable = TRUE
		SqlExecute.connectionIdent = Ident
		SqlExecute.pSqlStatement = ADR("EXEC Supertrack.uspWriteSequenceCount 0 , 2 ,1584")
		SqlExecute FUB dbExecuteSql()
		IF SqlExecute.status = ERR_OK THEN
			Sql = 2
		ENDIF
	ENDACTION

	ACTION 2:
		SqlDisconnect.enable = TRUE
		SqlDisconnect.connectionIdent = Ident
		SqlDisconnect FUB dbDisconnect()
		IF SqlDisconnect.status =  ERR_OK THEN
			Ident = 0
			Sql = 0
		ENDIF
	ENDACTION

	ACTION 3:
		SqlError.enable = TRUE
		SqlError.connectionIdent = Ident
		SqlError.pErrorMessage = ADR(ErrorString)
		SqlError.errorMessageSize = SIZEOF(ErrorString)
		SqlError FUB dbGetErrorMessage()
		IF SqlError.status = ERR_OK THEN
			Sql = 2
		ENDIF
	ENDACTION
ENDCASE

END_PROGRAM
```

### Test_bagMaint.var
```iecst
(********************************************************************
 * COPYRIGHT -- HP
 ********************************************************************
 * Program: Test_bagMaint
 * File: Test_bagMaint.var
 * Author: treamsbottom
 * Created: May 05, 2015
 ********************************************************************
 * Local variables of program Test_bagMaint
 ********************************************************************)
VAR
	TEST_STATE : INT;
	mySql : UINT;
	SqlWriteActive : BOOL;
	myBagNumber : STRING[5];
	myBagState : UINT;
	WaitReply : BOOL;
END_VAR
```

### zzGetNameSQL.typ
```iecst
(********************************************************************
 * COPYRIGHT --
 ********************************************************************
 * Package: TrackView
 * File: TrackView.typ
 * Author: Administrator
 * Created: March 02, 2009
 ********************************************************************
 * Data types of package TrackView
 ********************************************************************)

TYPE
	zzGetNamesTyp : 	STRUCT
		BagNumber : UINT;
		Prg : UDINT;
		PrgLong : STRING[8];
		PrgName : STRING[32];
		Cat : UDINT;
		CatLong : STRING[8];
		CatName : STRING[32];
		Cus : UDINT;
		CusLong : STRING[8];
		CusName : STRING[32];
		ImagePath : STRING[32];
		Description : STRING[10];
	END_STRUCT;
END_TYPE
```

### zzGetNameSQL.var
```iecst
(********************************************************************
 * COPYRIGHT --
 ********************************************************************
 * Package: TrackView
 * File: TrackView.var
 * Author: Dave Jefferys
 * Created: March 02, 2009
 ********************************************************************
 * Variables of package TrackView
 ********************************************************************)
VAR
	zzGetNamesData : ARRAY[0..39] OF zzGetNamesTyp;
END_VAR
```

### Program Logical/SQL/zzGetNamesSQL/zzGetNameSQL

#### zzGetNames.var
```iecst
(********************************************************************
 * COPYRIGHT --
 ********************************************************************
 * Program: zzGetNames
 * File: zzGetNames.var
 * Author: Dave
 * Created: November 19, 2010
 ********************************************************************
 * Local variables of program zzGetNames
 ********************************************************************)
VAR
	MaxDisplays : UINT;
	OwnerID : UDINT;
	TviewReplyOwnerID : UDINT;
	WaitReply : BOOL;
	myBag : UINT;
	CommsID : UDINT;
	Timer2Q : BOOL;
	Timer1Q : BOOL;
	Timer1ET : UDINT;
	Timer2ET : UDINT;
	result : DINT;
	TestTim : UDINT;
	mySql : UINT;
	myPrgString : STRING[24];
	myCatString : STRING[24];
	myCusString : STRING[24];
	SqlWriteActive : BOOL;
	RefreshDataTest : BOOL;
	n : INT;
END_VAR
```

#### zzGetNames.ab
```automation-basic
(********************************************************************
 * COPYRIGHT --
 ********************************************************************
 * Program: zzGetNames
 * File: zzGetNames.ab
 * Author: Dave
 * Created: November 19, 2010
 ********************************************************************
 * Implementation of program zzGetNames
 ********************************************************************)

;Get names from TrackView - Program, Category and Customer

;Version 1.00 19/11/2010 D.J. First Issue
;Version 2.00 12/12/2010 D.J. Added default values
;Version 3.00 19/10/2011 D.J. Clear Name when number has changed - if no TrackView then name will remain clear.

;Enter the required bag numbers for collection of names. Use the resulting names in transmisions to displays.

PROGRAM _INIT
	mySql = 96
	MaxDisplays = 1
	LOOP n = 1 TO MaxDisplays DO
		zzGetNamesData[n].BagNumber = 199 + n
	ENDLOOP
	;zzGetNamesData[20].BagNumber = 194	; Static Bag
	;zzGetNamesData[21].BagNumber = 411	; Customer Change 1
	;zzGetNamesData[22].BagNumber = 412	; Customer Change 2
	;zzGetNamesData[23].BagNumber = 401	; Customer Change Current Cust 1
	;zzGetNamesData[24].BagNumber = 402	; Customer Change Current Cust 2

	IF (MaxDisplays > SIZEOF(zzGetNamesData)) THEN
		MaxDisplays = SIZEOF(zzGetNamesData)
	ENDIF

	WaitReply = FALSE

	zzGetNamesData[0].BagNumber = 1
	zzGetNamesData[0].Prg		= 1
	strcpy(ADR(zzGetNamesData[0].PrgLong),"PRG")
	strcpy(ADR(zzGetNamesData[0].PrgName),"ProgramName")
	zzGetNamesData[0].Cat		= 1
	strcpy(ADR(zzGetNamesData[0].CatLong),"CAT")
	strcpy(ADR(zzGetNamesData[0].CatName),"CategoryName")
	zzGetNamesData[0].Cus		= 1
	strcpy(ADR(zzGetNamesData[0].CusLong),"CUS")
	strcpy(ADR(zzGetNamesData[0].CusName),"CustomerName")

END_PROGRAM

PROGRAM _CYCLIC
	IF RefreshDataTest THEN
		LOOP n = 1 TO MaxDisplays DO
			zzGetNamesData[n].Cat = 0
		ENDLOOP
		RefreshDataTest = FALSE
	ENDIF
	;Clear all display strings while waiting for replies,

	LOOP n = 1 TO MaxDisplays DO
		myBag = zzGetNamesData[n].BagNumber

		IF ((zzGetNamesData[n].Prg <> Bag[myBag].Prg) AND (Bag[myBag].Prg > 0)) THEN
			memcpy(ADR(zzGetNamesData[n].PrgLong),ADR(""),8)
			memcpy(ADR(zzGetNamesData[n].PrgName),ADR(""),32)
		ENDIF

		IF ((zzGetNamesData[n].Cat <> Bag[myBag].Cat) AND (Bag[myBag].Cat > 0)) THEN
			memcpy(ADR(zzGetNamesData[n].CatLong),ADR(""),8)
			memcpy(ADR(zzGetNamesData[n].CatName),ADR(""),32)
		ENDIF

		IF ((zzGetNamesData[n].Cus <> Bag[myBag].Cus) AND (Bag[myBag].Cus > 0)) THEN
			memcpy(ADR(zzGetNamesData[n].CusLong),ADR(""),8)
			memcpy(ADR(zzGetNamesData[n].CusName),ADR(""),32)
		ENDIF
	ENDLOOP

	;Search for display data that needs updating
	IF NOT WaitReply THEN

		OwnerID = OwnerID + 1
		IF (OwnerID > MaxDisplays) THEN
			OwnerID = 1
		ENDIF

		myBag = zzGetNamesData[OwnerID].BagNumber

		IF ((zzGetNamesData[OwnerID].Prg <> Bag[myBag].Prg) AND (Bag[myBag].Prg > 0)) THEN
			memcpy(ADR(zzGetNamesData[OwnerID].PrgLong),ADR(""),8)
			memcpy(ADR(zzGetNamesData[OwnerID].PrgName),ADR(""),32)
			WaitReply = TRUE
		ENDIF

		IF ((zzGetNamesData[OwnerID].Cat <> Bag[myBag].Cat) AND (Bag[myBag].Cat > 0)) THEN
			;Special for Brolli Get Prg code back for Data entry
			IF ((OwnerID = 25) OR (OwnerID = 26)) THEN
				Bag[myBag].Prg = 0
				zzGetNamesData[OwnerID].Prg = 0
				memcpy(ADR(zzGetNamesData[OwnerID].PrgLong),ADR(""),8)
				memcpy(ADR(zzGetNamesData[OwnerID].PrgName),ADR(""),32)
			ENDIF
			memcpy(ADR(zzGetNamesData[OwnerID].CatLong),ADR(""),8)
			memcpy(ADR(zzGetNamesData[OwnerID].CatName),ADR(""),32)
			WaitReply = TRUE
		ELSE IF Bag[myBag].Cat = 0 THEN
			zzGetNamesData[OwnerID].Cat = 0
			strcpy(ADR(zzGetNamesData[OwnerID].CatLong),"")
			strcpy(ADR(zzGetNamesData[OwnerID].CatName),"")
			strcpy(ADR(zzGetNamesData[OwnerID].CusName),"")
			strcpy(ADR(zzGetNamesData[OwnerID].PrgName),"")
			strcpy(ADR(zzGetNamesData[OwnerID].ImagePath),"")
		ENDIF

		IF ((zzGetNamesData[OwnerID].Cus <> Bag[myBag].Cus) AND (Bag[myBag].Cus > 0)) THEN
			memcpy(ADR(zzGetNamesData[OwnerID].CusLong),ADR(""),8)
			memcpy(ADR(zzGetNamesData[OwnerID].CusName),ADR(""),32)
			WaitReply = TRUE
		ENDIF

		;Set TrackView Registers
		IF WaitReply THEN
			itoa(Bag[myBag].Prg,ADR(myPrgString))
			itoa(Bag[myBag].Cat,ADR(myCatString))
			itoa(Bag[myBag].Cus,ADR(myCusString))
			SqlRequest[mySql].Request = TRUE
		ENDIF

	ENDIF

	;Set request to TrackView until reply
	IF (WaitReply AND SqlRequest[mySql].Complete) THEN

		myBag = zzGetNamesData[OwnerID].BagNumber

		strcpy(ADR(zzGetNamesData[OwnerID].PrgLong),ADR(SqlRequest[mySql].OutputData[1]))
		strcpy(ADR(zzGetNamesData[OwnerID].PrgName),ADR(SqlRequest[mySql].OutputData[2]))
		result = strcmp(ADR(zzGetNamesData[OwnerID].PrgName),"ProgCodeReturned")
		IF (result = 0) THEN
			Bag[myBag].Prg = USINT(atoi(ADR(zzGetNamesData[OwnerID].PrgLong)))
		ENDIF
		zzGetNamesData[OwnerID].Prg = Bag[myBag].Prg

		zzGetNamesData[OwnerID].Cat = Bag[myBag].Cat
		strcpy(ADR(zzGetNamesData[OwnerID].CatLong),ADR(SqlRequest[mySql].OutputData[3]))
		strcpy(ADR(zzGetNamesData[OwnerID].CatName),ADR(SqlRequest[mySql].OutputData[4]))

		zzGetNamesData[OwnerID].Cus = Bag[myBag].Cus
		strcpy(ADR(zzGetNamesData[OwnerID].CusLong),ADR(SqlRequest[mySql].OutputData[5]))
		strcpy(ADR(zzGetNamesData[OwnerID].CusName),ADR(SqlRequest[mySql].OutputData[6]))

		strcpy(ADR(zzGetNamesData[OwnerID].ImagePath),ADR(SqlRequest[mySql].OutputData[7]))

		WaitReply 	= FALSE

	ENDIF

IF SqlRequest[mySql].Request AND NOT SqlWriteActive THEN ; Write Count to SQL
	SqlWriteActive = TRUE
	SqlRequest[mySql].SQLType = cSQLType_ReadWrite
	SqlRequest[mySql].SQL_usp = cSQLReq_zzGetNames
	SqlRequest[mySql].NoOfParams = 3

	SqlRequest[mySql].Parameters[0].Type = cSQLParam_Input ;PLC Stn
	strcpy(ADR(SqlRequest[mySql].Parameters[0].Param_String),ADR(myPrgString))
	SqlRequest[mySql].Parameters[1].Type = cSQLParam_Input ;BatchID;
	strcpy(ADR(SqlRequest[mySql].Parameters[1].Param_String),ADR(myCatString))
	SqlRequest[mySql].Parameters[2].Type = cSQLParam_Input ; Prg
	strcpy(ADR(SqlRequest[mySql].Parameters[2].Param_String),ADR(myCusString))
ENDIF

IF SqlRequest[mySql].Complete THEN ; ClearRequest
	;Copy Out Reply Done in step.!
	SqlRequest[mySql] = cEmptySQlReq
	SqlWriteActive = FALSE
ELSE IF SqlRequest[mySql].Fail THEN
	WaitReply = FALSE ; Move to next and try and again
	SqlWriteActive = FALSE ; Reload Parameters
	SqlRequest[mySql].Fail = FALSE
;ELSE IF WaitReply AND NOT SqlWriteActive THEN
;	WaitReply = FALSE
ENDIF

END_PROGRAM
```

### zzSQL_Lib.typ
```iecst
(********************************************************************
 * COPYRIGHT -- HP
 ********************************************************************
 * Library: zzSQL_Lib
 * File: zzSQL_Lib.typ
 * Author: treamsbottom
 * Created: May 04, 2012
 ********************************************************************
 * Data types of library zzSQL_Lib
 ********************************************************************)

TYPE
	zzSQLGetNameTyp : 	STRUCT
		BagNumber : UINT;
		Prg : UDINT;
		PrgLong : STRING[8];
		PrgName : STRING[32];
		Cat : UDINT;
		CatLong : STRING[8];
		CatName : STRING[32];
		Cus : UDINT;
		CusLong : STRING[8];
		CusName : STRING[32];
	END_STRUCT;
	SQL_Enum :
		(
		eError,
		eConnect,
		eReadData,
		eDisconnect,
		eExecute,
		eGetData,
		eColumnCount,
		eGetAffectedRow,
		eIdle
		);
	SQLRequest_typ : 	STRUCT
		SQLType : USINT; (**Read Only - Write*)
		SQL_usp : USINT; (**Where in index is SQL usp cmd*)
		RequestID : UDINT; (**ID Used to return Results*)
		Complete : BOOL; (**Reponse when Complete*)
		NoOfParams : USINT; (**Number of Parameters*)
		Parameters : ARRAY[0..19]OF SQL_Parameter;
		Request : BOOL;
		OutputData : ARRAY[0..Dec_SqlOutputTypArrayLen]OF SQL_Output;
		Fail : BOOL;
	END_STRUCT;
	SQL_Typ : 	STRUCT
		Login : SQLLogin_typ;
	END_STRUCT;
	SQLLogin_typ : 	STRUCT
		Path : STRING[64];
		DBName : STRING[64];
		User : STRING[64];
		Password : STRING[64];
	END_STRUCT;
	SQL_Parameter : 	STRUCT
		Type : USINT; (**Input = 0 or Output = 1*)
		Param_String : STRING[32];
	END_STRUCT;
	SQL_Output :STRING[32];
END_TYPE
```

### Constants.var
```iecst
(********************************************************************
 * COPYRIGHT -- HP
 ********************************************************************
 * Package: NewPackage
 * File: Constants.var
 * Author: treamsbottom
 * Created: October 01, 2013
 ********************************************************************
 * Variables of package NewPackage
 ********************************************************************)
VAR CONSTANT
	dec_c_MaxSQL : USINT := 99;
	cSQLType_WriteOnly : USINT := 0;
	cSQLType_ReadWrite : USINT := 1;
	cSQLType_ReadOnly : USINT := 2;
	SQL_Port : STRING[5] := ':1433';
	cSQL_Comma_Space : STRING[2] := ', ';
	cSQL_Space : STRING[1] := ' ';
	cEmptySQlReq : SQLRequest_typ := (0); (**Used to clear buffer - like bag[0]*)
	cSQLParam_Input : USINT := 0;
	cSQLParam_Output : USINT := 1;
END_VAR
(**Constants for Sql Commands*)
VAR CONSTANT
	cSqluspCommands : ARRAY[0..19] OF STRING[50] := ['EXEC Supertrack.uspWriteSequenceCount','','EXEC Supertrack.uspBatchCreate','EXEC Supertrack.uspBatchUpdate','EXEC Supertrack.uspBatchVerify','EXEC Supertrack.uspBatchVerifyWithDelete','','EXEC Supertrack.uspBatchVerifyDeleteRetState','EXEC Supertrack.uspPicDBGetFTPPathPLC','EXEC Supertrack.uspzzGetNames','EXEC Supertrack.uspMaintenanceBagCount','EXEC Supertrack.uspMaintenanceBagGetState','EXEC Supertrack.uspMaintenanceBagCountReplyState','EXEC Supertrack.uspzzGetMultiNames',6('')]; (**Array of all Stored Procedure Strings*)
	cSQLReq_WriteSeqCount : USINT := 0;
	cSQLReq_BatchCreate : USINT := 2;
	cSQLReq_BatchUpdate : USINT := 3;
	cSQLReq_BatchVerify : USINT := 4;
	cSQLReq_BatchVerifyWithDelete : USINT := 5;
	cSQLReq_BatchVerifyDeleteReState : USINT := 7;
	cSQLReq_PicDBGetFTPPathPLC : USINT := 8;
	cSQLReq_zzGetNames : USINT := 9;
	cSQLReq_BagMaintCount : USINT := 10; (** Send count value to Maintenance DB PARAMS @PLC, @BAG*)
	cSQLReq_BagMaintGetState : USINT := 11; (** Read bag maintenance state @PLC, @BAG, @STATE*)
	cSQLReq_BagMaintCount_R_State : USINT := 12; (** Send count value and read bag maintenance state  @PLC, @BAG, @STATE*)
	cSQLReq_zzGetMultiNames : USINT := 13;
END_VAR
(*-*Constant Return Values for Batch Verify*)
VAR CONSTANT
	cSQL_BatchVerfiy_Match : USINT := 1;
	cSQL_BatchVerfiy_MisMatch : USINT := 2;
	cSQL_BatchVerfiy_DoesntExist : USINT := 3;
END_VAR
```

### zzSQL_Lib.var
```iecst
(********************************************************************
 * COPYRIGHT -- HP
 ********************************************************************
 * Library: zzSQL_Lib
 * File: zzSQL_Lib.var
 * Author: treamsbottom
 * Created: May 04, 2012
 ********************************************************************
 * Constants of library zzSQL_Lib
 ********************************************************************)
VAR CONSTANT
	Dec_SqlOutputTypArrayLen : USINT := 19;
END_VAR
```

- Program Logical/SQL/zzSQLDriver (IEC, version 1.00.1) (no source held here)

### zzTvText.var
```iecst
(********************************************************************
 * COPYRIGHT -- HP
 ********************************************************************
 * Program: zzTviewText
 * File: zzTviewText.var
 * Author: Dave
 * Created: January 30, 2013
 ********************************************************************
 * Local variables of program zzTviewText
 ********************************************************************)
VAR CONSTANT
	SendSUPDBServer : UDINT := 1;
	SendSUPDBName : UDINT := 2;
	SendSUPDBLogin : UDINT := 3;
	SendSUPDBPword : UDINT := 4;
	StartSQLServerDataRead : UDINT := 101;
	StartReadTextwords : UDINT := 102;
	SendTextWord : UDINT := 1000;
END_VAR
VAR
	myTviewString : STRING[64];
	myRequest : UDINT;
	StartRequest : BOOL;
	TviewRequest : UDINT;
	StartSQLServerRead : BOOL;
	StartTextwords : BOOL;
	Login : STRING[6];
	result : DINT;
END_VAR
```

### Global.typ
```iecst
TYPE
	Alm : 	STRUCT
		On : BOOL;
		Bag : UINT;
		ET : TIME;
		InList : BOOL;
		Name : UINT;
		Extra : UINT;
		Beacon : BOOL;
		Time : UDINT;
	END_STRUCT;
	BagType : 	STRUCT
		Cat : USINT;
		Dst : USINT;
		Wgt : UINT;
		Cnt : UINT;
		Cus : UINT;
		Day : USINT;
		Spare : USINT;
	END_STRUCT;
	CardInputs : 	STRUCT
		X01 : BOOL;
		X02 : BOOL;
		X03 : BOOL;
		X04 : BOOL;
		X05 : BOOL;
		X06 : BOOL;
		X07 : BOOL;
		X08 : BOOL;
		X09 : BOOL;
		X10 : BOOL;
		X11 : BOOL;
		X12 : BOOL;
		X13 : BOOL;
		X14 : BOOL;
		X15 : BOOL;
		X16 : BOOL;
	END_STRUCT;
	CardOutputs : 	STRUCT
		Y01 : BOOL;
		Y02 : BOOL;
		Y03 : BOOL;
		Y04 : BOOL;
		Y05 : BOOL;
		Y06 : BOOL;
		Y07 : BOOL;
		Y08 : BOOL;
		Y09 : BOOL;
		Y10 : BOOL;
		Y11 : BOOL;
		Y12 : BOOL;
		Y13 : BOOL;
		Y14 : BOOL;
		Y15 : BOOL;
		Y16 : BOOL;
	END_STRUCT;
	DAM : 	STRUCT
		Alive : UINT;
		Analog : INT;
	END_STRUCT;
	Enable_Vars : 	STRUCT
		Search : UINT;
		TransferBelt : BOOL;
		Ongoing : ARRAY[0..4]OF BOOL;
		Offgoing : ARRAY[0..4]OF BOOL;
		SBS : ARRAY[0..4]OF BOOL;
		SLU : ARRAY[0..9]OF BOOL;
		SIC : ARRAY[0..9]OF BOOL;
		SDC : ARRAY[0..9]OF BOOL;
		SPI : ARRAY[0..9]OF BOOL;
		SPN : ARRAY[0..9]OF BOOL;
		SVC : ARRAY[0..9]OF BOOL;
		SWB : ARRAY[0..4]OF BOOL;
		SPF : ARRAY[0..1]OF BOOL;
		SLU1 : BOOL;
		SVC2 : BOOL;
	END_STRUCT;
	Line_Vars : 	STRUCT
		Clear : BOOL;
		Full : BOOL;
		Trip : BOOL;
		FirstBag : UINT;
		LastBag : UINT;
		Space : UINT;
		SpaceBIT : UINT;
	END_STRUCT;
	Loading_Vars : 	STRUCT
		StartStn : UINT;
		EndStn : UINT;
		EnableStnRelease : BOOL;
		BeltHasRun : BOOL;
		Found : UINT;
		Line : UINT;
		Search : UINT;
	END_STRUCT;
	ReadDisplay : 	STRUCT
		Data : ARRAY[0..7]OF USINT;
	END_STRUCT;
	Reports : 	STRUCT
		Cat : UINT;
		Cus : UINT;
		Wgt : UINT;
		Cnt : UINT;
		Stn : UINT;
		Mcn : UINT;
	END_STRUCT;
	Request_Vars : 	STRUCT
		SDC1 : BOOL;
		SDC2 : BOOL;
		SDC2Full : BOOL;
		SIC1 : BOOL;
		SPF : BOOL;
		SVC1 : BOOL;
		TransferBelt : BOOL;
	END_STRUCT;
	ScanTime : 	STRUCT
		Start : TIME;
		End : TIME;
		Time : UINT;
		Min : UINT;
		Max : UINT;
	END_STRUCT;
	Std_Vars : 	STRUCT
		HaltSys : BOOL;
		HaltSysLoading : BOOL;
		StopSystem : BOOL;
		SafetyOn : BOOL;
		SafetyOnLoading : BOOL;
		AutoMaticRelease : BOOL;
		AutoRecirculation : BOOL;
		BagsWithDestinations : BOOL;
		BagsWithDestinations2 : BOOL;
		BagWithDestAtFront : BOOL;
		BagSpacing : USINT;
		Clock100ms : BOOL;
		Clock200ms : BOOL;
		Clock500ms : BOOL;
		Clock1s : BOOL;
		Clock2s : BOOL;
		EStop : BOOL;
		EStopLoading : BOOL;
		EnableOverUnderRelease : BOOL;
		MaxKanLink : USINT;
		MaxCats : USINT;
		MaxCust : UINT;
		MaxDischargers : USINT;
		MaxIO : UINT;
		MaxLines : UINT;
		MaxLinesBuffers : UINT;
		MaxWeighstations : UINT;
		MaxCountingStations : UINT;
		MaxStationBanks : UINT;
		MaxSearch : UINT;
		MinReleaseWeight : UINT;
		Monitor : UINT;
		MotorOverload : BOOL;
		MotorOverloadLoading : BOOL;
		PairingLoop : BOOL;
		Purging : BOOL;
		PurgeCompleted : BOOL;
		RepSpacing : USINT;
		StnBatchCode : UINT;
		StnsInQ : BOOL;
		StnsToPurge : BOOL;
		StationBagsStart : ARRAY[0..4]OF UINT;
		CountingBagsStart : UINT;
		StationReports : BOOL;
		StationsClosed : BOOL;
		TransferBeltRun : BOOL;
		UnloadingMaxDepth : UINT;
		CustomerFIFO : BOOL;
		CustomerFound : BOOL;
		AutoLineAllocation : BOOL;
		CustomerNewFound : BOOL;
		CustomerEditFound : BOOL;
	END_STRUCT;
	Stn_Mix : 	STRUCT
		Cat : ARRAY[0..9]OF UINT;
		Cus : ARRAY[0..9]OF UINT;
		Wgt : ARRAY[0..9]OF UINT;
		Cnt : ARRAY[0..9]OF UINT;
	END_STRUCT;
	Stn_Vars : 	STRUCT
		DestManual : UINT;
		LampOn : BOOL;
		ManualRelease : BOOL;
		QTime : UINT;
		ReleaseButton : BOOL;
		SpacesRequired : UINT;
		SP1 : BOOL;
		SP2 : BOOL;
		SP3 : BOOL;
		Count : UINT;
		Reg : UINT;
		Closed : BOOL;
		CntInput : BOOL;
		Weight : INT;
		Open : BOOL;
		PBCount : UINT;
		LampFlashFast : BOOL;
		CloseFlap : BOOL;
		Unlock : BOOL;
	END_STRUCT;
	Test_Vars : 	STRUCT
		TransferBelt : BOOL;
		Stations : BOOL;
		Dropped : ARRAY[0..4]OF BOOL;
		Drop : ARRAY[0..4]OF BOOL;
		Dischargers : BOOL;
	END_STRUCT;
	Uld_Vars : 	STRUCT
		SDCReady : BOOL;
		SDCSpaces : UINT;
		DischargerStartLine : UINT;
		LastCustQtyComplete : UINT;
		FIFOCustomer : UINT;
		FIFOCustomerFound : BOOL;
		FIFONextCustomer : UINT;
	END_STRUCT;
	WriteDisplay : 	STRUCT
		Data : ARRAY[0..7]OF USINT;
	END_STRUCT;
	comstype : 	STRUCT
		delime : UINT;
		delim : ARRAY[0..1]OF USINT;
		tx_cnt : UINT;
		rx_cnt : UINT;
		tx_len : UINT;
		rx_len : UINT;
		argc : UINT;
		argv : UDINT;
		idle : UINT;
	END_STRUCT;
	fiLOCAL_OBJ : 	STRUCT
		StateMan : UINT;
		ErrMan : UINT;
		Init : UDINT;
	END_STRUCT;
END_TYPE
```

### Global.var
```iecst
VAR RETAIN
	Alarm : ARRAY[0..109] OF Alm;
	AlarmBagNotProxLine : UINT;
	Bag : ARRAY[0..999] OF BagType;
	C : ARRAY[0..99] OF UINT;
	D : ARRAY[0..5999] OF UINT;
	Enable : Enable_Vars;
	Ldg : ARRAY[0..4] OF Loading_Vars;
	Line : ARRAY[0..99] OF Line_Vars;
	ReportBuffer : ARRAY[0..199] OF Reports;
	ReportLoading : ARRAY[0..50] OF Reports;
	ReportUnloading : ARRAY[0..10] OF Reports;
	Request : Enable_Vars;
	Std : Std_Vars;
	Stn : ARRAY[0..50] OF Stn_Vars;
	TCScan : ARRAY[0..8] OF ScanTime;
	Test : Test_Vars;
	Uld : ARRAY[0..20] OF Uld_Vars;
END_VAR
VAR CONSTANT
	almBagDataError : UINT := 20;
	almBagNotArrived : UINT := 6;
	almBagNotAtProx : UINT := 16;
	almBagNotReleased : UINT := 9;
	almBagNotSettled : UINT := 7;
	almEmergencyStop : UINT := 1;
	almGeneralSequence : UINT := 15;
	almInverterFault : UINT := 18;
	almLoadNotDropped : UINT := 10;
	almMotorOverload : UINT := 2;
	almNoAlarm : UINT := 0;
	almSwitchFault : UINT := 5;
END_VAR
VAR
	OK : ARRAY[0..40] OF BOOL;
END_VAR
VAR CONSTANT
	almUldNoBag : UINT := 4;
	almUldProgFinished : UINT := 3;
END_VAR
VAR
	AI354RAW_1 : INT; (* ±10 V, resolution 12 bit *)
	AI354RAW_2 : INT; (* ±10 V, resolution 12 bit *)
	AI354RAW_3 : INT; (* ±10 V, resolution 12 bit *)
	AI354RAW_4 : INT; (* ±10 V, resolution 12 bit *)
	I_EStop : BOOL;
	Indication : ARRAY[0..79] OF BOOL;
	SSS2Raw : DINT;
	SSS2Weight : UINT;
	SSS3Raw : DINT;
	SSS3Weight : UINT;
	SSS4Raw : DINT;
	AI2744Raw : ARRAY[0..20] OF DINT;
	SSS4Weight : UINT;
	StnPrev : ARRAY[0..50] OF BagType;
	TimerAlarm : TON_10ms;
	X : ARRAY[0..39] OF CardInputs;
	Y : ARRAY[0..39] OF CardOutputs;
	YForceDisable : ARRAY[0..39] OF CardOutputs;
	Zero : UINT := 0;
	pBag : UDINT;
	pC : UDINT;
	pD : UDINT;
END_VAR
```

- Program Logical/zztc2end (IEC, version 1.00.0) - * TC2 End - Scan Time Calculation (no source held here)

### Program Logical/zzclrmem (IEC) - * Clear Permanent Memory

#### zzclrmem.var
```iecst
VAR
	ClearMem	:BOOL;
	Dave	:UDINT;
END_VAR
```

### Program Logical/zzweigh (IEC) - * Station Weight Calculation and Calibration

#### zzweigh.var
```iecst
VAR RETAIN
	n : UINT;
	WeightUnits : DINT;
	StnHigh : UINT;
	StnLow : UINT;
	StnTestWgt : UINT;
	HighLow : UDINT;
	RawLow : DINT;
	StnRaw : ARRAY[0..99] OF UINT;
	NewLow : UINT;
	NewHigh : UINT;
END_VAR
VAR
	tstRaw : DINT;
	myRaw : DINT;
	myStnRaw : UINT;
	test : BOOL;
	w1 : UINT;
	w2 : UINT;
	w3 : UINT;
	w4 : UINT;
	UseAI2744 : BOOL;
END_VAR
```

#### zzweighCyclic.ab
```automation-basic
PROGRAM _CYCLIC
	(* cyclic program *)

;---------------------------------------------------------------------------------------------
;Revision 1.00 01/05/2001 D.J. First Issue
;Revision 2.00 23/10/2002 D.J. WeightUnits changed to DINT (problem when raw values over 32767
;Revision 3.00 22/08/2006 D.J. Changed for AI261
;---------------------------------------------------------------------------------------------

;------------------------------------------------------------
;WeighStation Calibration and Weight Calculation - With AI261
;------------------------------------------------------------
UseAI2744 = TRUE
;divide by 1000 should give around 50 parts per kg and keep raw value within UINT
;Add 32000 to value to ensure always positive
LOOP n = 1 TO Std.MaxWeighstations DO
	;To view a particular stn then set tstRaw to the required stn
	IF tstRaw > 0 THEN
		myRaw = tstRaw ;AI261Raw[tstRaw]
	ELSE
		myRaw = AI2744Raw[n]//????????????????????????????????????????????????
	ENDIF
	;Ensure raw value is within + 24bit if out of range + 32bit
	IF (myRaw = $7FFFFFFF) THEN
		myRaw = $FFFFFF
	ENDIF
	;Ensure raw value is within - 24bit if out of range - 32bit
	IF (myRaw = $80000001) THEN
		myRaw = $FF000001
	ENDIF
	;Convert raw to UINT the 3 least significant digits are removed
	IF UseAI2744 THEN
		myStnRaw = UINT((myRaw / 100) + 32000)
	ELSE
		myStnRaw = UINT((myRaw / 1000) + 32000)
	ENDIF
	StnRaw[n] = myStnRaw
ENDLOOP

LOOP n = 1 TO Std.MaxWeighstations DO

	StnLow 		= D[3400 + n]
	StnHigh 	= D[3500 + n]
	StnTestWgt 	= D[3600 + n]

	;Calibrate Low - From TrackView
	IF (D[995] = n) AND (D[996] = 11) THEN
		NewLow = StnRaw[n]
		IF (NewLow > 0) AND (NewLow < $FFFF) THEN
			D[3400 + n] = NewLow
		ENDIF
		D[996] = 0 ;Cancel the Cal-Low
	ENDIF
	;Calibrate High - From TrackView
	IF (D[995] = n) AND (D[996] = 12) AND (D[997] > 0) THEN
		NewHigh = StnRaw[n]
		IF (NewHigh > 0) AND (NewHigh < $FFFF) AND (NewHigh > StnLow) THEN
			D[3500 + n] = NewHigh
			D[3600 + n] = D[997]		;Test-Weight
		ENDIF
		D[996] = 0 ;Cancel the Cal-High
	ENDIF

	;Weigh Calculation - Multiply up to give accurate results
	HighLow = StnHigh - StnLow
	HighLow = HighLow * 1000
	;Avoid "Divide By Zero"
	IF (StnTestWgt > 0) THEN
		WeightUnits = DINT(HighLow / StnTestWgt)
		RawLow = INT(StnRaw[n] - StnLow)
		RawLow = RawLow * 1000
		IF (WeightUnits > 0) THEN ;AND (RawLow > 0) THEN
			Stn[n].Weight = INT(RawLow / WeightUnits)
		ELSE
			Stn[n].Weight = 0
		ENDIF
	ELSE
		Stn[n].Weight = 999
	ENDIF

ENDLOOP

IF test THEN
Stn[1].Weight = w1
Stn[2].Weight = w2
Stn[3].Weight = w3
Stn[4].Weight = w4
ENDIF
END_PROGRAM
```

- Program Logical/zzreport (IEC, version 1.00.0) - * Reports to Master PC (no source held here)

### Program Logical/zztime (IEC, version 1.00.0) - * System running time

#### zztimeInit.ab
```automation-basic
PROGRAM _INIT
(* init program *)

PLCFirstScan = TRUE
END_PROGRAM
```

### Package Logical/Mewa - Your Project Rename

### Package Logical/Mewa/200ms - 200ms Tasks

### Package Logical/Mewa/200ms/CAN - CAN Communication Variables

### can.typ
```iecst
TYPE
	CAN_Vars : 	STRUCT
		BagReady : BOOL;
		BatchCode : UINT;
		BatchID : UDINT;
		Category : UDINT;
		Customer : UDINT;
		Destination : UINT;
		DropLoad : BOOL;
		DoubleLoad : BOOL;
		Drier1Loading : BOOL;
		Drier2Loading : BOOL;
		Drier1Unloading : BOOL;
		Drier2Unloading : BOOL;
		FaultNumber : USINT;
		Live : BOOL;
		LiveTime : UINT;
		LoadDropped : BOOL;
		LoadFinished : BOOL;
		MachineID : UINT;
		Program : UINT;
		PressShift : BOOL;
		ReadyToLoad : BOOL;
		SP1 : UINT;
		SP2 : UINT;
		SP3 : UINT;
		StrobeComplete : BOOL;
		Transfer : BOOL;
		UnloadFinished : BOOL;
		Weight : UINT;
	END_STRUCT;
	WET_CAN : 	STRUCT
		ControlSignals : USINT;
		ControlSignals2 : USINT;
		Category : UINT;
		Customer : UINT;
		Weight : UINT;
	END_STRUCT;
	Box_CONTROL : 	STRUCT
		ControlSignals : USINT;
		Destination : USINT;
		Category : UINT;
		Weight : UINT;
		Spare : UINT;
	END_STRUCT;
	Box_CUS_BAT : 	STRUCT
		Customer : UDINT;
		BatchNumber : UDINT;
	END_STRUCT;
	Box_CUS_DST : 	STRUCT
		Customer : UDINT;
		Destination : USINT;
		Spare1 : USINT;
		Spare2 : USINT;
		Spare3 : USINT;
	END_STRUCT;
	Box_SP_CAT : 	STRUCT
		SP1 : UINT;
		SP2 : UINT;
		SP3 : UINT;
		Category : UINT;
	END_STRUCT;
END_TYPE
```

### Program Logical/Mewa/200ms/CAN/can_drv2 (IEC) - * PowerTrans 1 & 2

#### can_drv2.var
```iecst
VAR RETAIN
	CAN_enable : BOOL;
	ReadFrame1 : WET_CAN;
	EventRead1 : BOOL;
	EventWrite1 : BOOL;
	LastError : UINT;
	n : UINT;
	CANOK : BOOL;
	WriteFrame1 : WET_CAN;
	EventRead2 : BOOL;
	ReadFrame2 : WET_CAN;
	EventWrite2 : BOOL;
	WriteFrame2 : WET_CAN;
END_VAR
VAR
	CANopen_01 : CANopen;
	DOInfo : DatObjInfo;
	CANdftab_01 : CANdftab;
	error_var : UDINT;
	data_adr : UDINT;
	CANrwtab_01 : CANrwtab;
	Remainder : UINT;
	WgtRound : UINT;
	CanOff : BOOL;
	CanOffET : UDINT;
	CAN1 : BOOL;
END_VAR
```

#### can_drv2.ab
```automation-basic
;CAN Bus data exchange with CBW

;--------------------------------------------------------
;Version 1.00 02/11/2009 D.J. First Issue
;Version 2.00 22/04/2011 D.J. Weight Calculation now here
;--------------------------------------------------------

PROGRAM _INIT

CAN_enable = 1
EventWrite1 = 0									;Reset CAN data table WRITE event
EventRead1 = 0  								;Reset CAN data table READ event
EventWrite2 = 0									;Reset CAN data table WRITE event
EventRead2 = 0  								;Reset CAN data table READ event
;EventWrite3 = 0									;Reset CAN data table WRITE event
;EventRead3 = 0  							    ;Reset CAN data table READ event

CANopen_01.enable		= CAN_enable
CANopen_01.baud_rate	= 25					;Define baud rate - 250 kbit/s      CS1070 11= CAN H  21= CAN L 12 = CAN G
CANopen_01.cob_anz		= 100      				;Define number of link objects
CANopen_01.error_adr	= ADR(error_var)		;Define address for error output
CANopen_01.device		= ADR ("SL1.IF1.ST1.IF1.ST2.IF1")	;Define number of device ("SL1.IF1.ST1.IF1.ST2.IF1") ("SL1.IF1.ST1.IF1.ST2.IF1")   port on unit ("SL1.IF3") 5 = CAN H 6 = CANL 7= CAN GROUND
CANopen_01.info			= 0

CANopen_01 FUB CANopen()						;Initiate CANopen   SL1.IF1.ST1.IF1.ST2

IF CANopen_01.status=0 THEN						;Check error level

	DOInfo.enable = 1
	DOInfo.pName  = "can_cmd"

	DOInfo FUB DatObjInfo()

	IF (DOInfo.status = 0) THEN

		data_adr					= DOInfo.pDatObjMem
		CANdftab_01.enable			= 1
		CANdftab_01.us_ident 		= CANopen_01.us_ident	;Set us_id
		CANdftab_01.table_adr		= data_adr				;Define address of data object
		CANdftab_01.tab_num			= UINT(DOInfo.len / 72)	;Define number of values

		CANdftab_01 FUB CANdftab()    						;Initiate CANdftab

		IF CANdftab_01.status = 0 THEN
			WriteFrame1.ControlSignals = BIT_SET(WriteFrame1.ControlSignals,0);Set Live Signal
			WriteFrame2.ControlSignals = BIT_SET(WriteFrame2.ControlSignals,0)
			;WriteFrame3.ControlSignals = BIT_SET(WriteFrame3.ControlSignals,0)
			CANOK = TRUE
		ENDIF

	ENDIF

ENDIF

END_PROGRAM

PROGRAM _CYCLIC

IF CANOK THEN

	;----------------
	;Set Write values
	;----------------

	;------------------------------------------------------
	;Configure the CAN write to CBW1 SDC1
	;------------------------------------------------------

	IF CAN[1].BagReady THEN
		WriteFrame1.ControlSignals = BIT_SET(WriteFrame1.ControlSignals, 1)
	ELSE
		WriteFrame1.ControlSignals = BIT_CLR(WriteFrame1.ControlSignals, 1)
	ENDIF

	;WriteFrame1.FaultNumber = 0
	WriteFrame1.Category    = UINT(CAN[1].Category)
	WriteFrame1.Customer    = UINT(CAN[1].Customer)
	WriteFrame1.Weight      = CAN[1].Weight

	;Write to Machine1
	EventWrite1 = TRUE

	;WriteFrame1a.Machine    = CAN[1].MachineID
	;WriteFrame1a.BatchCode  = CAN[1].BatchCode
	;WriteFrame1a.Spare1 	= 0
	;WriteFrame1a.Spare2 	= 0

	;EventWrite1a = TRUE

	;------------------------------------------------------
	;Configure the CAN write to CBW2 SDC2
	;------------------------------------------------------
	IF CAN[2].BagReady THEN
			WriteFrame2.ControlSignals = BIT_SET(WriteFrame2.ControlSignals, 1)
	ELSE
			WriteFrame2.ControlSignals = BIT_CLR(WriteFrame2.ControlSignals, 1)
	ENDIF

	;WriteFrame2.FaultNumber = 0
	WriteFrame2.Category = UINT(CAN[2].Category)
	WriteFrame2.Customer 	= UINT(CAN[2].Customer)
	WriteFrame2.Weight 		= CAN[2].Weight

	;Write to CBW2
	EventWrite2 = TRUE

	;WriteFrame2a.Machine 	= CAN[2].MachineID
	;WriteFrame2a.BatchCode 	= CAN[2].BatchCode
	;WriteFrame2a.Spare1 	= 0
	;WriteFrame2a.Spare2 	= 0

	;EventWrite2a = TRUE

	;------------------------
	;Service CAN table
	;------------------------

	IF CANdftab_01.status=0 THEN						(*check error level*)
		CANrwtab_01.enable		= 1
		CANrwtab_01.tab_ident	= CANdftab_01.tab_ident (*define tab_id*)
		CANrwtab_01 FUB CANrwtab()						(*initiate CANrwtab*)
		LastError = CANrwtab_01.status
	ENDIF

	;----------------------------------------------------
	;Check for incomming data from CBW1
	;----------------------------------------------------
	IF EventRead1 = TRUE THEN
		EventRead1 = FALSE

		CAN[1].Live 		= BIT_TST(ReadFrame1.ControlSignals,0)
	;	CAN1							= BIT_TST(ReadFrame1.ControlSignals,0)
		CAN[1].DropLoad 	= BIT_TST(ReadFrame1.ControlSignals,1)
		CAN[1].LoadDropped 	= BIT_TST(ReadFrame1.ControlSignals,2)
		;CAN[1].FaultNumber	= ReadFrame1.FaultNumber

		IF CAN[1].Live THEN
			CAN[1].LiveTime = 50	;5 seconds
		ENDIF

		IF NOT CAN[1].Live THEN
			ReadFrame1.ControlSignals = BIT_CLR(ReadFrame1.ControlSignals,0)
		ENDIF

	ENDIF
	;CAN[1].Live = CAN1
	;----------------------------------------------------
	;Check for incomming data from CBW2
	;----------------------------------------------------
	IF EventRead2 = TRUE THEN
		EventRead2 = FALSE

		CAN[2].Live			= BIT_TST(ReadFrame2.ControlSignals,0)
		CAN[2].DropLoad		= BIT_TST(ReadFrame2.ControlSignals,1)
		CAN[2].LoadDropped  = BIT_TST(ReadFrame2.ControlSignals,2)
		;CAN[2].FaultNumber  = ReadFrame2.FaultNumber

		IF CAN[2].Live THEN
			CAN[2].LiveTime = 50	;5 seconds
		ENDIF

		IF NOT CAN[2].Live THEN
			ReadFrame2.ControlSignals = BIT_CLR(ReadFrame2.ControlSignals,0)
		ENDIF

	ENDIF
;	IF (CAN1) THEN
;		CAN[1].Live = TRUE
 ;   ENDIF
;TON_10ms(( NOT CAN1),200,CanOff,CanOffET)
;IF CanOff THEN
;	CAN[1].Live = FALSE
;ENDIF
	;-----------------
	;Live section
	;-----------------
	LOOP n = 1 TO 2 DO

		IF (CAN[n].LiveTime > 0) THEN
			CAN[n].LiveTime = (CAN[n].LiveTime - 1)
		ENDIF

;		CAN[n].Live = (CAN[n].LiveTime <> 0)

	ENDLOOP

ENDIF
IF (CAN[1].LiveTime >0) THEN
	CAN[1].Live = TRUE
ELSE
	CAN[1].Live = FALSE
ENDIF
IF (CAN[2].LiveTime >0) THEN
	CAN[2].Live = TRUE
ELSE
	CAN[2].Live = FALSE
ENDIF

;Monitor Registers for TrackView
D[81] = UINT(ReadFrame1.ControlSignals)	;ID = 121
D[82] = UINT(WriteFrame1.ControlSignals)	;ID = 120

D[83] = UINT(ReadFrame2.ControlSignals)	;ID = 131
D[84] = UINT(WriteFrame2.ControlSignals)	;ID = 130

;D[85] = UINT(ReadFrame3.ControlSignals)	;ID = 141
;D[86] = UINT(WriteFrame3.ControlSignals)	;ID = 140

;D[87] = UINT(ReadFrame4.ControlSignals)	;ID = 261
;D[88] = UINT(WriteFrame4.ControlSignals)	;ID = 260

;D[89] = UINT(ReadFrame5.ControlSignals)	;ID = 251
;D[90] = UINT(WriteFrame5.ControlSignals)	;ID = 241

;D[91] = UINT(ReadFrame6.ControlSignals)	;ID = 252
;D[92] = UINT(WriteFrame6.ControlSignals)	;ID = 242

;D[93] = UINT(ReadFrame7.ControlSignals)	;ID = 253
;D[94] = UINT(WriteFrame7.ControlSignals)	;ID = 243

;D[95] = UINT(ReadFrame8.ControlSignals)	;ID = 254
;D[96] = UINT(WriteFrame8.ControlSignals)	;ID = 244

END_PROGRAM
```

### Data object Logical/Mewa/200ms/CAN/can_cmd (Simple, version 2.00.0) - * Powertrans 1 & 2

#### can_cmd.dat
```
;-----------------
;CAN Command Table
;-----------------

;----------------------------------------------------------------------------------------
;Version 2.00 16/08/2011 D.J. Added task name to variables required by AR 3.xx and higher
;----------------------------------------------------------------------------------------

;         1234567890123456789012345678901   1234567890123456789012345678901
00000121,"can_drv2:ReadFrame1            ","can_drv2:EventRead1            ",$00000000
00000120,"can_drv2:WriteFrame1           ","can_drv2:EventWrite1           ",$00000001

00000131,"can_drv2:ReadFrame2            ","can_drv2:EventRead2            ",$00000000
00000130,"can_drv2:WriteFrame2           ","can_drv2:EventWrite2           ",$00000001

;00000141,"can_drv2:ReadFrame3            ","can_drv2:EventRead3            ",$00000000
;00000140,"can_drv2:WriteFrame3           ","can_drv2:EventWrite3           ",$00000001
;   |          |                                 |                               |
; CAN ADR  Variable Name 31 Chrs             Event Variable 31 Chrs           Read = 0 Write = 1
```

### Program Logical/Mewa/200ms/CAN/can_stn (IEC, version 1.00.0) - * Sorting station and Suction boxes
